(* IEC 61131-3 sources: Mizera_Tube/Plc (part 5) *)

(* ---- usrCh8.plc ---- *)
*******************************************************************************
*******************************************************************************
*   @@@ CH8: Unload machine management
*******************************************************************************
*******************************************************************************
#funcdec "assi.plc"
#funcdec "cnc.plc"

#include "usrMem.inc"

VAR_IN_OUT
#include "mem.inc"
END_VAR

VAR
#include "cnc.inc"

GESTCH8:            GESTCH;
CH8END:             GESTCHEND;
GESTAX70:           GESTAX;
GESTAX71:           GESTAX;                         * Saw Following Support
GESTAX72:           GESTAX;
GESTAX73:           GESTAX;
GESTAX74:           GESTAX;
GESTAX75:           GESTAX;
AXLSREF71:          AX_LS_REF;
AXLSREF72:          AX_LS_REF;
AXLSREF73:          AX_LS_REF;
AXLSREF74:          AX_LS_REF;
AXLSREF75:          AX_LS_REF;

RTRIG_AX_SEL71:     R_TRIG;
RTRIG_AX_SEL72:     R_TRIG;
RTRIG_AX_SEL73:     R_TRIG;
RTRIG_AX_SEL74:     R_TRIG;
RTRIG_AX_SEL75:     R_TRIG;

UnSupp_71_GoUp:    BOOL;
UnSupp_72_GoUp:    BOOL;
UnSupp_73_GoUp:    BOOL;
UnSupp_74_GoUp:    BOOL;
UnSupp_75_GoUp:    BOOL;

END_VAR

#include "iol.inc"

VAR_IN_OUT
#include "usrIol.inc"
ActualQtaAbsRef     AT %pa18;                       * Absolute homing quota
QtaRefAbsSet        AT %LsPlc50;                    * Absolute homing quota setting
END_VAR

FUNCTION CH8

PATH %cn8

LD   ALWAYS_ONE                                     ** PLCFLAGS.1  Flag sempre stato on
ST   GESTCH8.xCmdFromInput

LD   ALWAYS_ONE                                     ** PLCFLAGS.1  Flag sempre stato on
ST   GESTCH8.xEscOpCmd

LD   %PLCFLAGS.0
ST   GESTCH8.xSelFromInput                          * Disabilita selezioni standard macchina

LD   Ch0_Ref_Gen
ST   GESTCH8.xSelREF

LD   Ch0_Ref_Sin
ST   GESTCH8.xSingleRef

LD   Ch0_Jog
ST   GESTCH8.xSelJOG

LD   Ch0_Inc
ST   GESTCH8.xSelINC

LD   Ch0_Auto
ST   GESTCH8.xSelAUT

LD   ProgRunCh0
ANDN %cn0.rc8.1
ANDN PlcEmerGen                                     ** M0.10 Emergenza generale
OR (
LD   Start_Ch0
AND  ch8_in_ref
)
OR(
LD   Start_Ch0
AND  BCI_MDI                                        ** rc0.11  Selettore modi operativi su MDI (semiautom)
AND (
 LD  UP_SELCHAN                                     ** ui17 Canale selezionato da monitor canale
 EQ  8
)
)
ST   GESTCH8.xStart                                 * comando START al canale (esterno)

LD   ResetChannels
ST   GESTCH8.xReset                                 * comando RESET al canale (esterno)

LD   %cn0.rc8.1                                    ** Condizioni richiesta hold canale 0
OR(
LD   Pul_Stop_Req
AND  BCI_MDI                                        ** rc0.11  Selettore modi operativi su MDI (semiautom)
)
ST   GESTCH8.xHold                                  * comando Hold al canale (esterno)

LD   Ch0Alarm
ST   GESTCH8.xEmer                                  * comando Emergenza al canale (esterno)

LD   8888
ST   GESTCH8.xPPNumber                              * numero part program da eseguire

LD   %PLCFLAGS.0
ST   GESTCH8.xBlkSearch
ST   GESTCH8.xIntBlkSrc                             * Forzam. esec. ricerca blocco interna
ST   GESTCH8.xOverstore                             * Ab. overstore dopo ricerca blocco (provv.)

LD   MainChFeedrate                                 ** feedrate for channel
ST   GESTCH8.xOverride

CAL  GESTCH8

LD   GESTCH8.yProgramRun                            * Programma in corso
ST   PRGRUN_CN8

LD   BCO_STB_GET                                    ** rc8.17 Strobe per GET resources
AND  AxStopSincGRPMacc                              ** (gPlc13.11)Assi Fermi per sincronismo GRP[ax]
ST   BCI_ACK_GET                                    ** rc0.29  ACK per GET resource

********************************************************************************
* Unload axes
********************************************************************************
* Virtual Axis(70)

LD  %cc1.0                                          * Maschera assi associata al canale 8
JMPCN noAx70

PATH %ax70

LD   ALWAYS_ZERO
ST   GESTAX70.xJogPlus

LD   ALWAYS_ZERO
ST   GESTAX70.xJogMinus

LD   ALWAYS_ONE
ST   GESTAX70.xZeroForced                           * Forzamento asse tarato

LD   ALWAYS_ZERO
ST   GESTAX70.xHoldMoving                           * Richiesta blocco avanzamento

LD   Res_Axes                                       ** (gPlc25.1) reset axes disable electric shaft
ST   GESTAX70.xUnlock

LDN  ch8_in_ref                                     ** channel 3 in ref
ST   GESTAX70.xEnFIR                                * Abilita filtri FIR
ST   GESTAX70.xEnFrComp                             ** Abilita friction compensation

LD   ALWAYS_ZERO                                    ** PLCFLAGS.0  Flag sempre stato off
ST   GESTAX70.xDisLimiter

LD   GESTAX50_xCloseLoop
ST   GESTAX70.xCloseLoop

LD   %cn0.rc8.3                                     * ch0 in alarm
OR   %cn3.rc8.3                                     * ch3 in alarm
**OR   EmerINC
ST   GESTAX70.xSetAlarm                             ** Forzamento allarme asse

CAL  GESTAX70

noAx70:

********************************************************************************
* Unload Support for Saw Cutting (71)
********************************************************************************
PATH %ax71
PATH %ax_lsref71

***************************************
*   POWER ON (PON)
***************************************
LD   %pa3.31                                        * Simulato
ORN  %cc1.1                                         * Maschera assi associata al canale
OR(
LD   %nvel11                                        ** 3,4=CANopen, Ecat
EQ   3
)
OR(
LD   %nvel11                                        ** 3,4=CANopen, Ecat
EQ   4
)
ST   Pon_UnSupp_71                                  ** PON unload support axis
***************************************

LDN  %ra3.2                                         * ra3.2  Direzione moto asse avanti
OR   %ra0.9                                         * ra0.9 Comando indietro
AND  %ra3.13                                        * ra3.13  Ordine di moto
ST   UnSupp_71_GoUp

LD  %cc1.1                                          * Maschera assi associata al canale 8
JMPCN NOAX71

***
*   LIMIT SWITCH & REFERENCE SWITCH

LD   %lsrefmode
ST   AXLSREF71.x_REF_mode                           * 0=use ref switch...

LD   %lsreflevel
ST   AXLSREF71.x_TYPE_LS                            * (1=NC, 0=NO)

LD   I_I_FC_L1_NEG
ST   AXLSREF71.x_MIN_LS                             * Min Limit switch

LD   I_I_FC_L1_POS                * C saw minimumm limit switchV
ST   AXLSREF71.x_MAX_LS                             * Max Limit switch

LD   ALWAYS_ZERO
ST   AXLSREF71.x_REF_S                              * Reference switch

CAL  AXLSREF71

LD   AXLSREF71.y_MIN_LS                             * Min Limit switch
ST   GESTAX71.xMinusLS                              * Negative limit switch

LD   AXLSREF71.y_MAX_LS                             * Max Limit switch
ST   GESTAX71.xPlusLS                               * Positive limit switch

LD   AXLSREF71.y_REF_S                              * Reference switch
ST   GESTAX71.xRefLS                                * Reference
***

LD   MainAxesPowerAllowed
AND  MainAxesPower                                  * PON
ST   GESTAX71.xCloseLoop

LD   GstMaccSelYCh8
ST   GESTAX71.xSelected

***************************************
* Change REF quota for ABS reference
***************************************
CAL  RTRIG_AX_SEL71(CLK:=GESTAX71.xSelected)

LD   RTRIG_AX_SEL71.Q
JMPCN NoSel71
LD   ActualQtaAbsRef                                ** Absolute homing quota
ST   QtaRefAbsSet                                   ** Absolute homing quota setting
NoSel71:

LD   GESTAX71.xSelected
AND  %nvel14.0                                      * Se Vale 1 ?gestito "Encoder Assoluto" (Da Configura Asse)
AND (
LD   ActualQtaAbsRef                                ** Absolute homing quota
NE   QtaRefAbsSet                                   ** Absolute homing quota setting
)
JMPCN NoEq71

LD   QtaRefAbsSet                                   ** Absolute homing quota setting
ST   ActualQtaAbsRef                                ** Absolute homing quota
NoEq71:
***************************************

LD   Pul_Jogp                                       ** (gPlc0.4)jog+ pushbutton
AND  GESTAX71.xSelected
ANDN PlcEmerGen                                     ** M0.10 Emergenza generale
AND  GESTAX71.xCloseLoop
ST   GESTAX71.xJogPlus

LD   Pul_Jogm                                       ** (gPlc0.5)jog- pushbutton
AND  GESTAX71.xSelected
ANDN PlcEmerGen                                     ** M0.10 Emergenza generale
AND  GESTAX71.xCloseLoop
ANDN CMD_HOLDMOVING_CH8.1
ST   GESTAX71.xJogMinus

LD   %nvel14.0                                      * Se Vale 1 ?gestito "Encoder Assoluto" (Da Configura Asse)
ST   GESTAX71.xZeroForced                           * Forzamento asse tarato

LD   GESTAX2_xHoldMoving                            * Richiesta blocco avanzamento
OR   CMD_HOLDMOVING_CH8.1                           ** M203 Hold moving command axis CH5 (bit0=X, bit1=Y...)
ST   GESTAX71.xHoldMoving                           * Richiesta blocco avanzamento

LD   Res_Axes                                       ** (gPlc25.1) reset axes disable electric shaft
ST   GESTAX71.xUnlock

LDN  ch8_in_ref                                     ** channel 3 in ref
ST   GESTAX71.xEnFIR                                * Abilita filtri FIR
ST   GESTAX71.xEnFrComp                             ** Abilita friction compensation

LD   ALWAYS_ZERO                                    ** PLCFLAGS.0  Flag sempre stato off
ST   GESTAX71.xDisLimiter

LD   %cn0.rc8.3                                     * ch0 in alarm
OR   %cn3.rc8.3                                     * ch3 in alarm
**OR   EmerINC
ST   GESTAX71.xSetAlarm                             ** Forzamento allarme asse

LD   usrReqGrantSup1
ST   GESTAX71.xFromPlc

CAL  GESTAX71

LD   GESTAX71.yDriveNotEn
S    %PLCerr3.0                                     * Axis 71, drive not enable

LD   BSG_INC                                        ** rg1.2 Selezione modo INC (inc.fissi)
JMPCN SVIX71

LD   %pa59                                          * Velocit?di Repos
MUL  1000
DIV  60
MUL  MainChFeedrate                                 ** (gPlc16) feed degli assi (%)
DIV  100
ST   %ra50                                          * Limitazione velocita' massima interpolazione

SVIX71:
NOAX71:

********************************************************************************
* Unload Support 1 (ax72)
********************************************************************************
PATH %ax72
PATH %ax_lsref72

***************************************
*   POWER ON (PON)
***************************************
LD   %pa3.31            * Simulato
ORN  %cc1.2             * Maschera assi associata al canale
OR(
LD   %nvel11            ** 3,4=CANopen, Ecat
EQ   3
)
OR(
LD   %nvel11            ** 3,4=CANopen, Ecat
EQ   4
)
ST   Pon_UnSupp_72      ** PON unload support axis
***************************************

LDN  %ra3.2                                         * ra3.2  Direzione moto asse avanti
OR   %ra0.9                                         * ra0.9 Comando indietro
AND  %ra3.13                                        * ra3.13  Ordine di moto
ST   UnSupp_72_GoUp

LD  %cc1.2           * Maschera assi associata al canale 8
JMPCN NOAX72

***
*   LIMIT SWITCH & REFERENCE SWITCH

LD   %lsrefmode
ST   AXLSREF72.x_REF_mode        * 0=use ref switch...

LD   %lsreflevel
ST   AXLSREF72.x_TYPE_LS         * (1=NC, 0=NO)

LD   I_I_FC_L2_NEG
ST   AXLSREF72.x_MIN_LS          * Min Limit switch

LD   I_I_FC_L2_POS               * C saw maximun limit switch
ST   AXLSREF72.x_MAX_LS          * Max Limit switch

LD   ALWAYS_ZERO
ST   AXLSREF72.x_REF_S           * Reference switch

CAL  AXLSREF72

LD   AXLSREF72.y_MIN_LS          * Min Limit switch
ST   GESTAX72.xMinusLS           * Negative limit switch

LD   AXLSREF72.y_MAX_LS          * Max Limit switch
ST   GESTAX72.xPlusLS            * Positive limit switch

LD   AXLSREF72.y_REF_S           * Reference switch
ST   GESTAX72.xRefLS             * Reference
***

LD   MainAxesPowerAllowed
AND  MainAxesPower               * PON
ST   GESTAX72.xCloseLoop

LD   GstMaccSelZCh8
ST   GESTAX72.xSelected

***************************************
* Change REF quota for ABS reference
***************************************
CAL  RTRIG_AX_SEL72(CLK:=GESTAX72.xSelected)

LD   RTRIG_AX_SEL72.Q
JMPCN NoSel72
LD   ActualQtaAbsRef               ** Absolute homing quota
ST   QtaRefAbsSet                  ** Absolute homing quota setting
NoSel72:

LD   GESTAX72.xSelected
AND  %nvel14.0                     * Se Vale 1 � gestito "Encoder Assoluto" (Da Configura Asse)
AND (
LD   ActualQtaAbsRef               ** Absolute homing quota
NE   QtaRefAbsSet                  ** Absolute homing quota setting
)
JMPCN NoEq72

LD   QtaRefAbsSet                  ** Absolute homing quota setting
ST   ActualQtaAbsRef               ** Absolute homing quota
NoEq72:
***************************************

LD   Pul_Jogp                      ** (gPlc0.4)jog+ pushbutton
AND  GESTAX72.xSelected
ANDN PlcEmerGen                      ** M0.10 Emergenza generale
AND  GESTAX72.xCloseLoop
ST   GESTAX72.xJogPlus

LD   Pul_Jogm                      ** (gPlc0.5)jog- pushbutton
AND  GESTAX72.xSelected
ANDN PlcEmerGen                      ** M0.10 Emergenza generale
AND  GESTAX72.xCloseLoop
ANDN CMD_HOLDMOVING_CH8.2
ST   GESTAX72.xJogMinus

LD   %nvel14.0                     * Se Vale 1 � gestito "Encoder Assoluto" (Da Configura Asse)
ST   GESTAX72.xZeroForced          * Forzamento asse tarato

LD   GESTAX2_xHoldMoving           * Richiesta blocco avanzamento
OR   CMD_HOLDMOVING_CH8.2          ** M203 Hold moving command axis CH5 (bit0=X, bit1=Y...)
ST   GESTAX72.xHoldMoving          * Richiesta blocco avanzamento

LD   Res_Axes                      ** (gPlc25.1) reset axes disable electric shaft
ST   GESTAX72.xUnlock

LDN  ch8_in_ref                    ** channel 3 in ref
ST   GESTAX72.xEnFIR               * Abilita filtri FIR
ST   GESTAX72.xEnFrComp            ** Abilita friction compensation

LD   ALWAYS_ZERO                   ** PLCFLAGS.0  Flag sempre stato off
ST   GESTAX72.xDisLimiter

LD   %cn0.rc8.3                    * ch0 in alarm
OR   %cn3.rc8.3                    * ch3 in alarm
ST   GESTAX72.xSetAlarm            ** Forzamento allarme asse

LD   usrReqGrantSup2
ST   GESTAX72.xFromPlc

CAL  GESTAX72

LD   GESTAX72.yDriveNotEn
S    %PLCerr3.1                    * Axis 72, drive not enable

LD   BSG_INC                       ** rg1.2 Selezione modo INC (inc.fissi)
JMPCN SVIX72

LD   %pa59                         * Velocit� di Repos
MUL  1000
DIV  60
MUL  MainChFeedrate                ** (gPlc16) feed degli assi (%)
DIV  100
ST   %ra50                         * Limitazione velocita' massima interpolazione

SVIX72:
NOAX72:

********************************************************************************
* Unload Support 2 (ax73)
********************************************************************************
PATH %ax73
PATH %ax_lsref73

***************************************
*   POWER ON (PON)
***************************************
LD   %pa3.31                                        * Simulato
ORN  %cc1.3                                         * Maschera assi associata al canale
OR(
LD   %nvel11                                        ** 3,4=CANopen, Ecat
EQ   3
)
OR(
LD   %nvel11                                        ** 3,4=CANopen, Ecat
EQ   4
)
ST   Pon_UnSupp_73                                  ** PON unload support axis
***************************************

LDN  %ra3.2                                         * ra3.2  Direzione moto asse avanti
OR   %ra0.9                                         * ra0.9 Comando indietro
AND  %ra3.13                                        * ra3.13  Ordine di moto
ST   UnSupp_73_GoUp

LD  %cc1.3                                          * Maschera assi associata al canale 8
JMPCN NOAX73

***
*   LIMIT SWITCH & REFERENCE SWITCH

LD   %lsrefmode
ST   AXLSREF73.x_REF_mode                           * 0=use ref switch...

LD   %lsreflevel
ST   AXLSREF73.x_TYPE_LS                            * (1=NC, 0=NO)

LD   I_I_FC_L3_NEG
ST   AXLSREF73.x_MIN_LS                             * Min Limit switch

LD   I_I_FC_L3_POS                                  * W maximun limit switch
ST   AXLSREF73.x_MAX_LS                             * Max Limit switch

LD   ALWAYS_ZERO
ST   AXLSREF73.x_REF_S                              * Reference switch

CAL  AXLSREF73

LD   AXLSREF73.y_MIN_LS                             * Min Limit switch
ST   GESTAX73.xMinusLS                              * Negative limit switch

LD   AXLSREF73.y_MAX_LS                             * Max Limit switch
ST   GESTAX73.xPlusLS                               * Positive limit switch

LD   AXLSREF73.y_REF_S                              * Reference switch
ST   GESTAX73.xRefLS                                * Reference
***

LD   MainAxesPowerAllowed
AND  MainAxesPower                                  * PON
ST   GESTAX73.xCloseLoop

LD   GstMaccSelUCh8
ST   GESTAX73.xSelected

***************************************
* Change REF quota for ABS reference
***************************************
CAL  RTRIG_AX_SEL73(CLK:=GESTAX73.xSelected)

LD   RTRIG_AX_SEL73.Q
JMPCN NoSel73
LD   ActualQtaAbsRef                                ** Absolute homing quota
ST   QtaRefAbsSet                                   ** Absolute homing quota setting
NoSel73:

LD   GESTAX73.xSelected
AND  %nvel14.0                                      * Se Vale 1 ?gestito "Encoder Assoluto" (Da Configura Asse)
AND (
LD   ActualQtaAbsRef                                ** Absolute homing quota
NE   QtaRefAbsSet                                   ** Absolute homing quota setting
)
JMPCN NoEq73

LD   QtaRefAbsSet                                   ** Absolute homing quota setting
ST   ActualQtaAbsRef                                ** Absolute homing quota
NoEq73:
***************************************

LD   Pul_Jogp                                       ** (gPlc0.4)jog+ pushbutton
AND  GESTAX73.xSelected
ANDN PlcEmerGen                                     ** M0.10 Emergenza generale
AND  GESTAX73.xCloseLoop
ST   GESTAX73.xJogPlus

LD   Pul_Jogm                                       ** (gPlc0.5)jog- pushbutton
AND  GESTAX73.xSelected
ANDN PlcEmerGen                                     ** M0.10 Emergenza generale
AND  GESTAX73.xCloseLoop
ANDN CMD_HOLDMOVING_CH8.3
ST   GESTAX73.xJogMinus

LD   %nvel14.0                                      * Se Vale 1 ?gestito "Encoder Assoluto" (Da Configura Asse)
ST   GESTAX73.xZeroForced                           * Forzamento asse tarato

LD   GESTAX2_xHoldMoving                            * Richiesta blocco avanzamento
OR  CMD_HOLDMOVING_CH8.3                           ** M203 Hold moving command axis CH5 (bit0=X, bit1=Y...)
ST   GESTAX73.xHoldMoving                           * Richiesta blocco avanzamento

LD   Res_Axes                                       ** (gPlc25.1) reset axes disable electric shaft
ST   GESTAX73.xUnlock

LDN  ch8_in_ref                                     ** channel 3 in ref
ST   GESTAX73.xEnFIR                                * Abilita filtri FIR
ST   GESTAX73.xEnFrComp                             ** Abilita friction compensation

LD   ALWAYS_ZERO                                    ** PLCFLAGS.0  Flag sempre stato off
ST   GESTAX73.xDisLimiter

LD   %cn0.rc8.3                                     * ch0 in alarm
OR   %cn3.rc8.3                                     * ch3 in alarm
**OR   EmerINC
ST   GESTAX73.xSetAlarm                             ** Forzamento allarme asse

LD   usrReqGrantSup3
ST   GESTAX73.xFromPlc

CAL  GESTAX73

LD   GESTAX73.yDriveNotEn
S    %PLCerr3.2                                     * Axis 73, drive not enable

LD   BSG_INC                                        ** rg1.2 Selezione modo INC (inc.fissi)
JMPCN SVIX73

LD   %pa59                                          * Velocit?di Repos
MUL  1000
DIV  60
MUL  MainChFeedrate                                 ** (gPlc16) feed degli assi (%)
DIV  100
ST   %ra50                                          * Limitazione velocita' massima interpolazione

SVIX73:
NOAX73:

********************************************************************************
* Unload Support 3 (ax74)
********************************************************************************
PATH %ax74
PATH %ax_lsref74

***************************************
*   POWER ON (PON)
***************************************
LD   %pa3.31                                        * Simulato
ORN  %cc1.4                                         * Maschera assi associata al canale
OR(
LD   %nvel11                                        ** 3,4=CANopen, Ecat
EQ   3
)
OR(
LD   %nvel11                                        ** 3,4=CANopen, Ecat
EQ   4
)
ST   Pon_UnSupp_74                                  ** PON unload support axis
***************************************

LDN  %ra3.2                                         * ra3.2  Direzione moto asse avanti
OR   %ra0.9                                         * ra0.9 Comando indietro
AND  %ra3.13                                        * ra3.13  Ordine di moto
ST   UnSupp_74_GoUp

LD  %cc1.4                                          * Maschera assi associata al canale 8
JMPCN NOAX74

***
*   LIMIT SWITCH & REFERENCE SWITCH

LD   %lsrefmode
ST   AXLSREF74.x_REF_mode                           * 0=use ref switch...

LD   %lsreflevel
ST   AXLSREF74.x_TYPE_LS                            * (1=NC, 0=NO)

LD   I_I_FC_L4_NEG
ST   AXLSREF74.x_MIN_LS                             * Min Limit switch

LD   I_I_FC_L4_POS                                  * W minimumm limit switch
ST   AXLSREF74.x_MAX_LS                             * Max Limit switch

LD   ALWAYS_ZERO
ST   AXLSREF74.x_REF_S                              * Reference switch

CAL  AXLSREF74

LD   AXLSREF74.y_MIN_LS                             * Min Limit switch
ST   GESTAX74.xMinusLS                              * Negative limit switch

LD   AXLSREF74.y_MAX_LS                             * Max Limit switch
ST   GESTAX74.xPlusLS                               * Positive limit switch

LD   AXLSREF74.y_REF_S                              * Reference switch
ST   GESTAX74.xRefLS                                * Reference
***

LD   MainAxesPowerAllowed
AND  MainAxesPower                                  * PON
ST   GESTAX74.xCloseLoop

LD   GstMaccSelVCh8
ST   GESTAX74.xSelected

***************************************
* Change REF quota for ABS reference
***************************************
CAL  RTRIG_AX_SEL74(CLK:=GESTAX74.xSelected)

LD   RTRIG_AX_SEL74.Q
JMPCN NoSel74
LD   ActualQtaAbsRef                                ** Absolute homing quota
ST   QtaRefAbsSet                                   ** Absolute homing quota setting
NoSel74:

LD   GESTAX74.xSelected
AND  %nvel14.0                                      * Se Vale 1 ?gestito "Encoder Assoluto" (Da Configura Asse)
AND (
LD   ActualQtaAbsRef                                ** Absolute homing quota
NE   QtaRefAbsSet                                   ** Absolute homing quota setting
)
JMPCN NoEq74

LD   QtaRefAbsSet                                   ** Absolute homing quota setting
ST   ActualQtaAbsRef                                ** Absolute homing quota
NoEq74:
***************************************

LD   Pul_Jogp                                       ** (gPlc0.4)jog+ pushbutton
AND  GESTAX74.xSelected
ANDN PlcEmerGen                                     ** M0.10 Emergenza generale
AND  GESTAX74.xCloseLoop
ST   GESTAX74.xJogPlus

LD   Pul_Jogm                                       ** (gPlc0.5)jog- pushbutton
AND  GESTAX74.xSelected
ANDN PlcEmerGen                                     ** M0.10 Emergenza generale
AND  GESTAX74.xCloseLoop
ANDN CMD_HOLDMOVING_CH8.4
ST   GESTAX74.xJogMinus

LD   %nvel14.0                                      * Se Vale 1 ?gestito "Encoder Assoluto" (Da Configura Asse)
ST   GESTAX74.xZeroForced                           * Forzamento asse tarato

LD   GESTAX2_xHoldMoving                            * Richiesta blocco avanzamento
OR   CMD_HOLDMOVING_CH8.4                           ** M203 Hold moving command axis CH5 (bit0=X, bit1=Y...)
ST   GESTAX74.xHoldMoving                           * Richiesta blocco avanzamento

LD   Res_Axes                                       ** (gPlc25.1) reset axes disable electric shaft
ST   GESTAX74.xUnlock

LDN  ch8_in_ref                                     ** channel 3 in ref
ST   GESTAX74.xEnFIR                                * Abilita filtri FIR
ST   GESTAX74.xEnFrComp                             ** Abilita friction compensation

LD   ALWAYS_ZERO                                    ** PLCFLAGS.0  Flag sempre stato off
ST   GESTAX74.xDisLimiter

LD   %cn0.rc8.3                                     * ch0 in alarm
OR   %cn3.rc8.3                                     * ch3 in alarm
ST   GESTAX74.xSetAlarm                             ** Forzamento allarme asse

LD   usrReqGrantSup4
ST   GESTAX74.xFromPlc

CAL  GESTAX74

LD   GESTAX74.yDriveNotEn
S    %PLCerr3.3                                     * Axis 74, drive not enable

LD   BSG_INC                                        ** rg1.2 Selezione modo INC (inc.fissi)
JMPCN SVIX74

LD   %pa59                                          * Velocit?di Repos
MUL  1000
DIV  60
MUL  MainChFeedrate                                 ** (gPlc16) feed degli assi (%)
DIV  100
ST   %ra50                                          * Limitazione velocita' massima interpolazione

SVIX74:
NOAX74:

********************************************************************************
* Unload Support 4 (ax75)
********************************************************************************
PATH %ax75
PATH %ax_lsref75

***************************************
*   POWER ON (PON)
***************************************
LD   %pa3.31                                        * Simulato
ORN  %cc1.5                                         * Maschera assi associata al canale
OR(
LD   %nvel11                                        ** 3,4=CANopen, Ecat
EQ   3
)
OR(
LD   %nvel11                                        ** 3,4=CANopen, Ecat
EQ   4
)
ST   Pon_UnSupp_75                                  ** PON unload support axis
***************************************

LDN  %ra3.2                                         * ra3.2  Direzione moto asse avanti
OR   %ra0.9                                         * ra0.9 Comando indietro
AND  %ra3.13                                        * ra3.13  Ordine di moto
ST   UnSupp_75_GoUp

LD  %cc1.5                                          * Maschera assi associata al canale 8
JMPCN NOAX75

***
*   LIMIT SWITCH & REFERENCE SWITCH

LD   %lsrefmode
ST   AXLSREF75.x_REF_mode                           * 0=use ref switch...

LD   %lsreflevel
ST   AXLSREF75.x_TYPE_LS                            * (1=NC, 0=NO)

LD   I_I_FC_L5_NEG
ST   AXLSREF75.x_MIN_LS                             * Min Limit switch

LD   I_I_FC_L5_POS
ST   AXLSREF75.x_MAX_LS                             * Max Limit switch

LD   ALWAYS_ZERO
ST   AXLSREF75.x_REF_S                              * Reference switch

CAL  AXLSREF75

LD   AXLSREF75.y_MIN_LS                             * Min Limit switch
ST   GESTAX75.xMinusLS                              * Negative limit switch

LD   AXLSREF75.y_MAX_LS                             * Max Limit switch
ST   GESTAX75.xPlusLS                               * Positive limit switch

LD   AXLSREF75.y_REF_S                              * Reference switch
ST   GESTAX75.xRefLS                                * Reference
***

LD   MainAxesPowerAllowed
AND  MainAxesPower                                  * PON
ST   GESTAX75.xCloseLoop

LD   GstMaccSelWCh8
ST   GESTAX75.xSelected

***************************************
* Change REF quota for ABS reference
***************************************
CAL  RTRIG_AX_SEL75(CLK:=GESTAX75.xSelected)

LD   RTRIG_AX_SEL75.Q
JMPCN NoSel75
LD   ActualQtaAbsRef                                ** Absolute homing quota
ST   QtaRefAbsSet                                   ** Absolute homing quota setting
NoSel75:

LD   GESTAX75.xSelected
AND  %nvel14.0                                      * Se Vale 1 ?gestito "Encoder Assoluto" (Da Configura Asse)
AND (
LD   ActualQtaAbsRef                                ** Absolute homing quota
NE   QtaRefAbsSet                                   ** Absolute homing quota setting
)
JMPCN NoEq75

LD   QtaRefAbsSet                                   ** Absolute homing quota setting
ST   ActualQtaAbsRef                                ** Absolute homing quota
NoEq75:
***************************************

LD   Pul_Jogp                                       ** (gPlc0.4)jog+ pushbutton
AND  GESTAX75.xSelected
ANDN PlcEmerGen                                     ** M0.10 Emergenza generale
AND  GESTAX75.xCloseLoop
ST   GESTAX75.xJogPlus

LD   Pul_Jogm                                       ** (gPlc0.5)jog- pushbutton
AND  GESTAX75.xSelected
ANDN PlcEmerGen                                     ** M0.10 Emergenza generale
AND  GESTAX75.xCloseLoop
ANDN CMD_HOLDMOVING_CH8.5
ST   GESTAX75.xJogMinus

LD   %nvel14.0                                      * Se Vale 1 ?gestito "Encoder Assoluto" (Da Configura Asse)
ST   GESTAX75.xZeroForced                           * Forzamento asse tarato

LD   GESTAX2_xHoldMoving                           * Richiesta blocco avanzamento
OR   CMD_HOLDMOVING_CH8.5                           ** M203 Hold moving command axis CH5 (bit0=X, bit1=Y...)
ST   GESTAX75.xHoldMoving                           * Richiesta blocco avanzamento

LD   Res_Axes                                       ** (gPlc25.1) reset axes disable electric shaft
ST   GESTAX75.xUnlock

LDN  ch8_in_ref                                     ** channel 3 in ref
ST   GESTAX75.xEnFIR                                * Abilita filtri FIR
ST   GESTAX75.xEnFrComp                             ** Abilita friction compensation

LD   ALWAYS_ZERO                                    ** PLCFLAGS.0  Flag sempre stato off
ST   GESTAX75.xDisLimiter

LD   %cn0.rc8.3                                     * ch0 in alarm
OR   %cn3.rc8.3                                     * ch3 in alarm
**OR   EmerINC
ST   GESTAX75.xSetAlarm                             ** Forzamento allarme asse

LD   usrReqGrantSup5
ST   GESTAX75.xFromPlc

CAL  GESTAX75

LD   GESTAX75.yDriveNotEn
S    %PLCerr3.3                                     * Axis 75, drive not enable

LD   BSG_INC                                        ** rg1.2 Selezione modo INC (inc.fissi)
JMPCN SVIX75

LD   %pa59                                          * Velocit?di Repos
MUL  1000
DIV  60
MUL  MainChFeedrate                                 ** (gPlc16) feed degli assi (%)
DIV  100
ST   %ra50                                          * Limitazione velocita' massima interpolazione

SVIX75:
NOAX75:

**************************
* Acknowledg funzioni "M"
**************************
*
LD   %PLCFLAGS.0
ST   CH8END.xWaitMFun

CAL  CH8END

END_FUNCTION

(* ---- usrCh9.plc ---- *)
*******************************************************************************
*******************************************************************************
*   @@@ CH9: Lateral /Loader horizontal axes support
*******************************************************************************
*******************************************************************************
#funcdec "assi.plc"
#funcdec "cnc.plc"

#include "usrMem.inc"

VAR_IN_OUT
#include "mem.inc"
END_VAR

VAR
#include "cnc.inc"

GESTCH9:            GESTCH;
CH9END:             GESTCHEND;
GESTAX80:           GESTAX;    * virtual axes for following
GESTAX81:           GESTAX;
GESTAX82:           GESTAX;
GESTAX83:           GESTAX;
GESTAX84:           GESTAX;

AXLSREF81:          AX_LS_REF;
AXLSREF82:          AX_LS_REF;
AXLSREF83:          AX_LS_REF;
AXLSREF84:          AX_LS_REF;
AXLSREF85:          AX_LS_REF;

RTRIG_AX_SEL81:     R_TRIG;
RTRIG_AX_SEL82:     R_TRIG;
RTRIG_AX_SEL83:     R_TRIG;
RTRIG_AX_SEL84:     R_TRIG;
RTRIG_AX_SEL85:     R_TRIG;

UnSupp_81_GoUp:    BOOL;
UnSupp_82_GoUp:    BOOL;
UnSupp_83_GoUp:    BOOL;
UnSupp_84_GoUp:    BOOL;
UnSupp_85_GoUp:    BOOL;

END_VAR

#include "iol.inc"

VAR_IN_OUT
#include "usrIol.inc"
ActualQtaAbsRef     AT %pa18;                       * Absolute homing quota
QtaRefAbsSet        AT %LsPlc50;                    * Absolute homing quota setting

END_VAR

FUNCTION CH9

PATH %cn9

LD   ALWAYS_ONE                                     ** PLCFLAGS.1  Flag sempre stato on
ST   GESTCH9.xCmdFromInput

LD   ALWAYS_ONE                                     ** PLCFLAGS.1  Flag sempre stato on
ST   GESTCH9.xEscOpCmd

LD   %PLCFLAGS.0
ST   GESTCH9.xSelFromInput                          * Disabilita selezioni standard macchina

LD   Ch0_Ref_Gen
ST   GESTCH9.xSelREF

LD   Ch0_Ref_Sin
ST   GESTCH9.xSingleRef

LD   Ch0_Jog
ST   GESTCH9.xSelJOG

LD   Ch0_Inc
ST   GESTCH9.xSelINC

LD   Ch0_Auto
ST   GESTCH9.xSelAUT

LD   %PLCFLAGS.0                                    ** Condizioni richiesta hold canale 0
ST   GESTCH9.xStart                                 * comando START al canale (esterno)

LD   ResetChannels
ST   GESTCH9.xReset                                 * comando RESET al canale (esterno)

LD   %PLCFLAGS.0                                    ** Condizioni richiesta hold canale 0
OR(
LD   Pul_Stop_Req
AND  BCI_MDI                                        ** rc0.11  Selettore modi operativi su MDI (semiautom)
)
ST   GESTCH9.xHold                                  * comando Hold al canale (esterno)

LD   Ch0Alarm
ST   GESTCH9.xEmer                                  * comando Emergenza al canale (esterno)

LD   99999
ST   GESTCH9.xPPNumber                              * numero part program da eseguire

LD   %PLCFLAGS.0
ST   GESTCH9.xBlkSearch
ST   GESTCH9.xIntBlkSrc                             * Forzam. esec. ricerca blocco interna
ST   GESTCH9.xOverstore                             * Ab. overstore dopo ricerca blocco (provv.)

LD   MainChFeedrate                                 ** feedrate for channel
ST   GESTCH9.xOverride

CAL  GESTCH9

LD   GESTCH9.yProgramRun                            * Programma in corso
ST   PRGRUN_CN9

LD   BCO_STB_GET                                    ** rc8.17 Strobe per GET resources
AND  AxStopSincGRPMacc                              ** (gPlc13.11)Assi Fermi per sincronismo GRP[ax]
ST   BCI_ACK_GET                                    ** rc0.29  ACK per GET resource

********************************************************************************
* Unload axes
********************************************************************************
* Virtual Axis(70)

LD  %cc1.0                                          * Maschera assi associata al canale 8
JMPCN noAx80

PATH %ax80

LD   ALWAYS_ZERO
ST   GESTAX80.xJogPlus

LD   ALWAYS_ZERO
ST   GESTAX80.xJogMinus

LD   ALWAYS_ONE
ST   GESTAX80.xZeroForced                           * Forzamento asse tarato

LD   ALWAYS_ZERO
ST   GESTAX80.xHoldMoving                           * Richiesta blocco avanzamento

LD   Res_Axes                                       ** (gPlc25.1) reset axes disable electric shaft
ST   GESTAX80.xUnlock

LDN  ch9_in_ref                                     ** channel 3 in ref
ST   GESTAX80.xEnFIR                                * Abilita filtri FIR
ST   GESTAX80.xEnFrComp                             ** Abilita friction compensation

LD   ALWAYS_ZERO                                    ** PLCFLAGS.0  Flag sempre stato off
ST   GESTAX80.xDisLimiter

LD   GESTAX50_xCloseLoop
ST   GESTAX80.xCloseLoop

LD   %cn0.rc8.3                                     * ch0 in alarm
OR   %cn3.rc8.3                                     * ch3 in alarm
**OR   EmerINC
ST   GESTAX80.xSetAlarm                             ** Forzamento allarme asse

CAL  GESTAX80

noAx80:

********************************************************************************
* Unload Support for Saw Cutting (81) 2
********************************************************************************
PATH %ax81
PATH %ax_lsref81

***************************************
*   POWER ON (PON)
***************************************
LD   %pa3.31                                        * Simulato
ORN  %cc1.1                                         * Maschera assi associata al canale
OR(
LD   %nvel11                                        ** 3,4=CANopen, Ecat
EQ   3
)
OR(
LD   %nvel11                                        ** 3,4=CANopen, Ecat
EQ   4
)
ST   Pon_UnSupp_81                                  ** PON unload support axis
***************************************

LDN  %ra3.2                                         * ra3.2  Direzione moto asse avanti
OR   %ra0.9                                         * ra0.9 Comando indietro
AND  %ra3.13                                        * ra3.13  Ordine di moto
ST   UnSupp_81_GoUp

LD  %cc1.1                                          * Maschera assi associata al canale 8
JMPCN NOAX81

***
*   LIMIT SWITCH & REFERENCE SWITCH

LD   %lsrefmode
ST   AXLSREF81.x_REF_mode                           * 0=use ref switch...

LD   %lsreflevel
ST   AXLSREF81.x_TYPE_LS                            * (1=NC, 0=NO)

LD   I_I_FC_O1_NEG
ST   AXLSREF81.x_MIN_LS                             * Min Limit switch

LD   I_I_FC_O1_POS
ST   AXLSREF81.x_MAX_LS                             * Max Limit switch

LD   ALWAYS_ZERO
ST   AXLSREF81.x_REF_S                              * Reference switch

CAL  AXLSREF81

LD   AXLSREF81.y_MIN_LS                             * Min Limit switch
ST   GESTAX81.xMinusLS                              * Negative limit switch

LD   AXLSREF81.y_MAX_LS                             * Max Limit switch
ST   GESTAX81.xPlusLS                               * Positive limit switch

LD   AXLSREF81.y_REF_S                              * Reference switch
ST   GESTAX81.xRefLS                                * Reference
***

LD   MainAxesPowerAllowed
AND  MainAxesPower                                  * PON
ST   GESTAX81.xCloseLoop

LD   Sel_Y_Ch9
ST   GESTAX81.xSelected

***************************************
* Change REF quota for ABS reference
***************************************
CAL  RTRIG_AX_SEL81(CLK:=GESTAX81.xSelected)

LD   RTRIG_AX_SEL81.Q
JMPCN NoSel81
LD   ActualQtaAbsRef                                ** Absolute homing quota
ST   QtaRefAbsSet                                   ** Absolute homing quota setting
NoSel81:

LD   GESTAX81.xSelected
AND  %nvel14.0                                      * Se Vale 1 ?gestito "Encoder Assoluto" (Da Configura Asse)
AND (
LD   ActualQtaAbsRef                                ** Absolute homing quota
NE   QtaRefAbsSet                                   ** Absolute homing quota setting
)
JMPCN NoEq81

LD   QtaRefAbsSet                                   ** Absolute homing quota setting
ST   ActualQtaAbsRef                                ** Absolute homing quota
NoEq81:
***************************************

LD   Pul_Jogp                                       ** (gPlc0.4)jog+ pushbutton
AND  GESTAX81.xSelected
ANDN PlcEmerGen                                     ** M0.10 Emergenza generale
AND  GESTAX81.xCloseLoop
ST   GESTAX81.xJogPlus

LD   Pul_Jogm                                       ** (gPlc0.5)jog- pushbutton
AND  GESTAX81.xSelected
ANDN PlcEmerGen                                     ** M0.10 Emergenza generale
AND  GESTAX81.xCloseLoop
*ANDN CMD_HOLDMOVING_CH9.1
ST   GESTAX81.xJogMinus

LD   %nvel14.0                                      * Se Vale 1 ?gestito "Encoder Assoluto" (Da Configura Asse)
ST   GESTAX81.xZeroForced                           * Forzamento asse tarato

LD   GESTAX2_xHoldMoving                            * Richiesta blocco avanzamento
OR(
LD   CMD_HOLDMOVING_CH9.1                           ** M203 Hold moving command axis CH5 (bit0=X, bit1=Y...)
*AND  UnSupp_81_GoUp
)
ST   GESTAX81.xHoldMoving                           * Richiesta blocco avanzamento

LD   Res_Axes                                       ** (gPlc25.1) reset axes disable electric shaft
ST   GESTAX81.xUnlock

LDN  ch9_in_ref                                     ** channel 3 in ref
ST   GESTAX81.xEnFIR                                * Abilita filtri FIR
ST   GESTAX81.xEnFrComp                             ** Abilita friction compensation

LD   ALWAYS_ZERO                                    ** PLCFLAGS.0  Flag sempre stato off
ST   GESTAX81.xDisLimiter

LD   %cn0.rc8.3                                     * ch0 in alarm
OR   %cn3.rc8.3                                     * ch3 in alarm
**OR   EmerINC
ST   GESTAX81.xSetAlarm                             ** Forzamento allarme asse

LD   usrReqGrantSupLat1
ST   GESTAX81.xFromPlc

CAL  GESTAX81

LD   GESTAX81.yDriveNotEn
S    %PLCerr3.24

LD   BSG_INC                                        ** rg1.2 Selezione modo INC (inc.fissi)
JMPCN SVIX81

LD   %pa59                                          * Velocit?di Repos
MUL  1000
DIV  60
MUL  MainChFeedrate                                 ** (gPlc16) feed degli assi (%)
DIV  100
ST   %ra50                                          * Limitazione velocita' massima interpolazione

SVIX81:
NOAX81:

********************************************************************************
* Unload Support 1 (ax71)
********************************************************************************
PATH %ax82
PATH %ax_lsref82

***************************************
*   POWER ON (PON)
***************************************
LD   %pa3.31            * Simulato
ORN  %cc1.2             * Maschera assi associata al canale
OR(
LD   %nvel11            ** 3,4=CANopen, Ecat
EQ   3
)
OR(
LD   %nvel11            ** 3,4=CANopen, Ecat
EQ   4
)
ST   Pon_UnSupp_82      ** PON unload support axis
***************************************

LDN  %ra3.2                                         * ra3.2  Direzione moto asse avanti
OR   %ra0.9                                         * ra0.9 Comando indietro
AND  %ra3.13                                        * ra3.13  Ordine di moto
ST   UnSupp_82_GoUp

LD  %cc1.2           * Maschera assi associata al canale 8
JMPCN NOAX82

***
*   LIMIT SWITCH & REFERENCE SWITCH

LD   %lsrefmode
ST   AXLSREF82.x_REF_mode        * 0=use ref switch...

LD   %lsreflevel
ST   AXLSREF82.x_TYPE_LS         * (1=NC, 0=NO)

LD   I_I_FC_O2_NEG
ST   AXLSREF82.x_MIN_LS          * Min Limit switch

LD   I_I_FC_O2_POS
ST   AXLSREF82.x_MAX_LS          * Max Limit switch

LD   ALWAYS_ZERO
ST   AXLSREF82.x_REF_S           * Reference switch

CAL  AXLSREF82

LD   AXLSREF82.y_MIN_LS          * Min Limit switch
ST   GESTAX82.xMinusLS           * Negative limit switch

LD   AXLSREF82.y_MAX_LS          * Max Limit switch
ST   GESTAX82.xPlusLS            * Positive limit switch

LD   AXLSREF82.y_REF_S           * Reference switch
ST   GESTAX82.xRefLS             * Reference
***

LD   MainAxesPowerAllowed
AND  MainAxesPower               * PON
ST   GESTAX82.xCloseLoop

LD   Sel_Z_Ch9
ST   GESTAX82.xSelected

***************************************
* Change REF quota for ABS reference
***************************************
CAL  RTRIG_AX_SEL82(CLK:=GESTAX82.xSelected)

LD   RTRIG_AX_SEL82.Q
JMPCN NoSel72
LD   ActualQtaAbsRef               ** Absolute homing quota
ST   QtaRefAbsSet                  ** Absolute homing quota setting
NoSel72:

LD   GESTAX82.xSelected
AND  %nvel14.0                     * Se Vale 1 � gestito "Encoder Assoluto" (Da Configura Asse)
AND (
LD   ActualQtaAbsRef               ** Absolute homing quota
NE   QtaRefAbsSet                  ** Absolute homing quota setting
)
JMPCN NoEq82

LD   QtaRefAbsSet                  ** Absolute homing quota setting
ST   ActualQtaAbsRef               ** Absolute homing quota
NoEq82:
***************************************

LD   Pul_Jogp                      ** (gPlc0.4)jog+ pushbutton
AND  GESTAX82.xSelected
ANDN PlcEmerGen                      ** M0.10 Emergenza generale
AND  GESTAX82.xCloseLoop
ST   GESTAX82.xJogPlus

LD   Pul_Jogm                      ** (gPlc0.5)jog- pushbutton
AND  GESTAX82.xSelected
ANDN PlcEmerGen                      ** M0.10 Emergenza generale
AND  GESTAX82.xCloseLoop
*ANDN CMD_HOLDMOVING_CH9.2
ST   GESTAX82.xJogMinus

LD   %nvel14.0                     * Se Vale 1 � gestito "Encoder Assoluto" (Da Configura Asse)
ST   GESTAX82.xZeroForced          * Forzamento asse tarato

LD   GESTAX2_xHoldMoving           * Richiesta blocco avanzamento
OR(
LD   CMD_HOLDMOVING_CH9.2          ** M203 Hold moving command axis CH5 (bit0=X, bit1=Y...)
*AND  UnSupp_82_GoUp
)
ST   GESTAX82.xHoldMoving          * Richiesta blocco avanzamento

LD   Res_Axes                      ** (gPlc25.1) reset axes disable electric shaft
ST   GESTAX82.xUnlock

LDN  ch9_in_ref                    ** channel 3 in ref
ST   GESTAX82.xEnFIR               * Abilita filtri FIR
ST   GESTAX82.xEnFrComp            ** Abilita friction compensation

LD   ALWAYS_ZERO                   ** PLCFLAGS.0  Flag sempre stato off
ST   GESTAX82.xDisLimiter

LD   %cn0.rc8.3                    * ch0 in alarm
OR   %cn3.rc8.3                    * ch3 in alarm
**OR   EmerINC
ST   GESTAX82.xSetAlarm            ** Forzamento allarme asse

LD   usrReqGrantSupLat2
ST   GESTAX82.xFromPlc

CAL  GESTAX82

LD   GESTAX82.yDriveNotEn
S    %PLCerr3.25

LD   BSG_INC                       ** rg1.2 Selezione modo INC (inc.fissi)
JMPCN SVIX82

LD   %pa59                         * Velocit� di Repos
MUL  1000
DIV  60
MUL  MainChFeedrate                ** (gPlc16) feed degli assi (%)
DIV  100
ST   %ra50                         * Limitazione velocita' massima interpolazione

SVIX82:
NOAX82:

********************************************************************************
* Unload Support 2 (ax73)
********************************************************************************
PATH %ax83
PATH %ax_lsref83

***************************************
*   POWER ON (PON)
***************************************
LD   %pa3.31                                        * Simulato
ORN  %cc1.3                                         * Maschera assi associata al canale
OR(
LD   %nvel11                                        ** 3,4=CANopen, Ecat
EQ   3
)
OR(
LD   %nvel11                                        ** 3,4=CANopen, Ecat
EQ   4
)
ST   Pon_UnSupp_83                                  ** PON unload support axis
***************************************

LDN  %ra3.2                                         * ra3.2  Direzione moto asse avanti
OR   %ra0.9                                         * ra0.9 Comando indietro
AND  %ra3.13                                        * ra3.13  Ordine di moto
ST   UnSupp_83_GoUp

LD  %cc1.3                                          * Maschera assi associata al canale 8
JMPCN NOAX83

***
*   LIMIT SWITCH & REFERENCE SWITCH

LD   %lsrefmode
ST   AXLSREF83.x_REF_mode                           * 0=use ref switch...

LD   %lsreflevel
ST   AXLSREF83.x_TYPE_LS                            * (1=NC, 0=NO)

LD   I_I_FC_O3_NEG
ST   AXLSREF83.x_MIN_LS                             * Min Limit switch

LD   I_I_FC_O3_POS
ST   AXLSREF83.x_MAX_LS                             * Max Limit switch

LD   ALWAYS_ZERO
ST   AXLSREF83.x_REF_S                              * Reference switch

CAL  AXLSREF83

LD   AXLSREF83.y_MIN_LS                             * Min Limit switch
ST   GESTAX83.xMinusLS                              * Negative limit switch

LD   AXLSREF83.y_MAX_LS                             * Max Limit switch
ST   GESTAX83.xPlusLS                               * Positive limit switch

LD   AXLSREF83.y_REF_S                              * Reference switch
ST   GESTAX83.xRefLS                                * Reference
***

LD   MainAxesPowerAllowed
AND  MainAxesPower                                  * PON
ST   GESTAX83.xCloseLoop

LD   Sel_U_Ch9
ST   GESTAX83.xSelected

***************************************
* Change REF quota for ABS reference
***************************************
CAL  RTRIG_AX_SEL83(CLK:=GESTAX83.xSelected)

LD   RTRIG_AX_SEL83.Q
JMPCN NoSel83
LD   ActualQtaAbsRef                                ** Absolute homing quota
ST   QtaRefAbsSet                                   ** Absolute homing quota setting
NoSel83:

LD   GESTAX83.xSelected
AND  %nvel14.0                                      * Se Vale 1 ?gestito "Encoder Assoluto" (Da Configura Asse)
AND (
LD   ActualQtaAbsRef                                ** Absolute homing quota
NE   QtaRefAbsSet                                   ** Absolute homing quota setting
)
JMPCN NoEq83

LD   QtaRefAbsSet                                   ** Absolute homing quota setting
ST   ActualQtaAbsRef                                ** Absolute homing quota
NoEq83:
***************************************

LD   Pul_Jogp                                       ** (gPlc0.4)jog+ pushbutton
AND  GESTAX83.xSelected
ANDN PlcEmerGen                                     ** M0.10 Emergenza generale
AND  GESTAX83.xCloseLoop
ST   GESTAX83.xJogPlus

LD   Pul_Jogm                                       ** (gPlc0.5)jog- pushbutton
AND  GESTAX83.xSelected
ANDN PlcEmerGen                                     ** M0.10 Emergenza generale
AND  GESTAX83.xCloseLoop
*ANDN CMD_HOLDMOVING_CH9.3
ST   GESTAX83.xJogMinus

LD   %nvel14.0                                      * Se Vale 1 ?gestito "Encoder Assoluto" (Da Configura Asse)
ST   GESTAX83.xZeroForced                           * Forzamento asse tarato

LD   GESTAX2_xHoldMoving                            * Richiesta blocco avanzamento
OR(
LD   CMD_HOLDMOVING_CH9.3                           ** M203 Hold moving command axis CH5 (bit0=X, bit1=Y...)
*AND  UnSupp_83_GoUp
)
ST   GESTAX83.xHoldMoving                           * Richiesta blocco avanzamento

LD   Res_Axes                                       ** (gPlc25.1) reset axes disable electric shaft
ST   GESTAX83.xUnlock

LDN  ch9_in_ref                                     ** channel 3 in ref
ST   GESTAX83.xEnFIR                                * Abilita filtri FIR
ST   GESTAX83.xEnFrComp                             ** Abilita friction compensation

LD   ALWAYS_ZERO                                    ** PLCFLAGS.0  Flag sempre stato off
ST   GESTAX83.xDisLimiter

LD   %cn0.rc8.3                                     * ch0 in alarm
OR   %cn3.rc8.3                                     * ch3 in alarm
**OR   EmerINC
ST   GESTAX83.xSetAlarm                             ** Forzamento allarme asse

LD   usrReqGrantSupLat3
ST   GESTAX83.xFromPlc

CAL  GESTAX83

LD   GESTAX83.yDriveNotEn
S    %PLCerr3.26

LD   BSG_INC                                        ** rg1.2 Selezione modo INC (inc.fissi)
JMPCN SVIX83

LD   %pa59                                          * Velocit?di Repos
MUL  1000
DIV  60
MUL  MainChFeedrate                                 ** (gPlc16) feed degli assi (%)
DIV  100
ST   %ra50                                          * Limitazione velocita' massima interpolazione

SVIX83:
NOAX83:

********************************************************************************
* Unload Support 3 (ax74)
********************************************************************************
PATH %ax84
PATH %ax_lsref84

***************************************
*   POWER ON (PON)
***************************************
LD   %pa3.31                                        * Simulato
ORN  %cc1.4                                         * Maschera assi associata al canale
OR(
LD   %nvel11                                        ** 3,4=CANopen, Ecat
EQ   3
)
OR(
LD   %nvel11                                        ** 3,4=CANopen, Ecat
EQ   4
)
ST   Pon_UnSupp_84                                  ** PON unload support axis
***************************************

LDN  %ra3.2                                         * ra3.2  Direzione moto asse avanti
OR   %ra0.9                                         * ra0.9 Comando indietro
AND  %ra3.13                                        * ra3.13  Ordine di moto
ST   UnSupp_84_GoUp

LD  %cc1.4                                          * Maschera assi associata al canale 8
JMPCN NOAX84

***
*   LIMIT SWITCH & REFERENCE SWITCH

LD   %lsrefmode
ST   AXLSREF84.x_REF_mode                           * 0=use ref switch...

LD   %lsreflevel
ST   AXLSREF84.x_TYPE_LS                            * (1=NC, 0=NO)

LD   I_I_FC_O4_NEG
ST   AXLSREF84.x_MIN_LS                             * Min Limit switch

LD   I_I_FC_O4_POS
ST   AXLSREF84.x_MAX_LS                             * Max Limit switch

LD   ALWAYS_ZERO
ST   AXLSREF84.x_REF_S                              * Reference switch

CAL  AXLSREF84

LD   AXLSREF84.y_MIN_LS                             * Min Limit switch
ST   GESTAX84.xMinusLS                              * Negative limit switch

LD   AXLSREF84.y_MAX_LS                             * Max Limit switch
ST   GESTAX84.xPlusLS                               * Positive limit switch

LD   AXLSREF84.y_REF_S                              * Reference switch
ST   GESTAX84.xRefLS                                * Reference
***

LD   MainAxesPowerAllowed
AND  MainAxesPower                                  * PON
ST   GESTAX84.xCloseLoop

LD   Sel_V_Ch9
ST   GESTAX84.xSelected

***************************************
* Change REF quota for ABS reference
***************************************
CAL  RTRIG_AX_SEL84(CLK:=GESTAX84.xSelected)

LD   RTRIG_AX_SEL84.Q
JMPCN NoSel84
LD   ActualQtaAbsRef                                ** Absolute homing quota
ST   QtaRefAbsSet                                   ** Absolute homing quota setting
NoSel84:

LD   GESTAX84.xSelected
AND  %nvel14.0                                      * Se Vale 1 ?gestito "Encoder Assoluto" (Da Configura Asse)
AND (
LD   ActualQtaAbsRef                                ** Absolute homing quota
NE   QtaRefAbsSet                                   ** Absolute homing quota setting
)
JMPCN NoEq84

LD   QtaRefAbsSet                                   ** Absolute homing quota setting
ST   ActualQtaAbsRef                                ** Absolute homing quota
NoEq84:
***************************************

LD   Pul_Jogp                                       ** (gPlc0.4)jog+ pushbutton
AND  GESTAX84.xSelected
ANDN PlcEmerGen                                     ** M0.10 Emergenza generale
AND  GESTAX84.xCloseLoop
ST   GESTAX84.xJogPlus

LD   Pul_Jogm                                       ** (gPlc0.5)jog- pushbutton
AND  GESTAX84.xSelected
ANDN PlcEmerGen                                     ** M0.10 Emergenza generale
AND  GESTAX84.xCloseLoop
*ANDN CMD_HOLDMOVING_CH9.4
ST   GESTAX84.xJogMinus

LD   %nvel14.0                                      * Se Vale 1 ?gestito "Encoder Assoluto" (Da Configura Asse)
ST   GESTAX84.xZeroForced                           * Forzamento asse tarato

LD   GESTAX2_xHoldMoving                            * Richiesta blocco avanzamento
OR(
LD   CMD_HOLDMOVING_CH9.4                           ** M203 Hold moving command axis CH5 (bit0=X, bit1=Y...)
*AND  UnSupp_84_GoUp
)
ST   GESTAX84.xHoldMoving                           * Richiesta blocco avanzamento

LD   Res_Axes                                       ** (gPlc25.1) reset axes disable electric shaft
ST   GESTAX84.xUnlock

LDN  ch9_in_ref                                     ** channel 3 in ref
ST   GESTAX84.xEnFIR                                * Abilita filtri FIR
ST   GESTAX84.xEnFrComp                             ** Abilita friction compensation

LD   ALWAYS_ZERO                                    ** PLCFLAGS.0  Flag sempre stato off
ST   GESTAX84.xDisLimiter

LD   %cn0.rc8.3                                     * ch0 in alarm
OR   %cn3.rc8.3                                     * ch3 in alarm
**OR   EmerINC
ST   GESTAX84.xSetAlarm                             ** Forzamento allarme asse

LD   usrReqGrantSupLat4
ST   GESTAX84.xFromPlc

CAL  GESTAX84

LD   GESTAX84.yDriveNotEn
S    %PLCerr3.27

LD   BSG_INC                                        ** rg1.2 Selezione modo INC (inc.fissi)
JMPCN SVIX84

LD   %pa59                                          * Velocit?di Repos
MUL  1000
DIV  60
MUL  MainChFeedrate                                 ** (gPlc16) feed degli assi (%)
DIV  100
ST   %ra50                                          * Limitazione velocita' massima interpolazione

SVIX84:
NOAX84:

**************************
* Acknowledg funzioni "M"
**************************
*
LD   %PLCFLAGS.0
ST   CH9END.xWaitMFun

CAL  CH9END

END_FUNCTION

(* ---- usrCmd.plc ---- *)
*******************************************************************************
*   usrCnd.plc
*   ESAutomotion
*   LASER machine
*******************************************************************************
VAR_IN_OUT
#include "mem.inc"
#include "usrIol.inc"
END_VAR
#include "usrMem.inc"

FUNCTION COMMAND_TO_MAIN

*CH3
* Hold V axis

LD   Hold_U_Z1Supp
OR   Hold_U_Z2Supp
OR   Hold_U_Z3Supp
OR   Hold_U_Z4Supp
OR   Hold_U_Z5Supp
OR   Hold_U_SupUnHorAx85
OR   Hold_U_SupUnHorAx86
OR   Hold_U_SupUnHorAx87
OR   Hold_U_SupUnHorAx88
OR   M_HoldAx_V
ST   CMD_HOLDMOVING_CH3.4            ** M202 Hold moving command axis CH3 (bit0=X, bit1=Y...)

* Hold X-U
LD   Hold_U_Z1SuppLoad
OR   Hold_U_Z2SuppLoad
OR   Hold_U_Z3SuppLoad
OR   Hold_U_Z4SuppLoad
OR   HoldO1Ax30_HOR
OR   HoldO2Ax30_HOR
OR   HoldO3Ax30_HOR
OR   HoldO4Ax30_HOR
OR   %PLCmsg8.5
OR   M_HoldAx_U
ST   CMD_HOLDMOVING_CH3.0            ** M202 Hold moving command axis CH3 (bit0=X, bit1=Y...)

* CH8 (Unloader)

LD   HoldZ1Supp
ST   CMD_HOLDMOVING_CH8.1            ** M203 Hold moving command axis CH5 (bit0=X, bit1=Y...)

LD   HoldZ2Supp
ST   CMD_HOLDMOVING_CH8.2            ** M203 Hold moving command axis CH5 (bit0=X, bit1=Y...)

LD   HoldZ3Supp
ST   CMD_HOLDMOVING_CH8.3            ** M203 Hold moving command axis CH5 (bit0=X, bit1=Y...)

LD   HoldZ4Supp
ST   CMD_HOLDMOVING_CH8.4            ** M203 Hold moving command axis CH5 (bit0=X, bit1=Y...)

LD   HoldZ5Supp
ST   CMD_HOLDMOVING_CH8.5            ** M203 Hold moving command axis CH5 (bit0=X, bit1=Y...)

* CH5

* Grant Request

LD   usrReqGrantSupL1
ST   GRANT5.1

LD   usrReqGrantSupL2
ST   GRANT5.2

LD   usrReqGrantSupL3
ST   GRANT5.3

LD   usrReqGrantSupL4
ST   GRANT5.4

* Hold support axes

LD   HoldZ1SuppLoad
ST   CMD_HOLDMOVING_CH5.1

LD   HoldZ2SuppLoad
ST   CMD_HOLDMOVING_CH5.2

LD   HoldZ3SuppLoad
ST   CMD_HOLDMOVING_CH5.3

LD   HoldZ4SuppLoad
ST   CMD_HOLDMOVING_CH5.4

* Hold support Lateral axes

LD   HoldO1SuppLoad_LAT
ST   CMD_HOLDMOVING_CH9.1

LD   HoldO2SuppLoad_LAT
ST   CMD_HOLDMOVING_CH9.2

LD   HoldO3SuppLoad_LAT
ST   CMD_HOLDMOVING_CH9.3

LD   HoldO4SuppLoad_LAT
ST   CMD_HOLDMOVING_CH9.4

*
END_FUNCTION

(* ---- usrGen.plc ---- *)
#include "iol.inc"
#include "usrMem.inc"

VAR
TON36:                TON;
appoggio:             BOOL;
State_AutOrg:         BOOL;
CurrState:            DWORD;
DangerThresld:        DWORD;
YZatParking:          DWORD;
emercaseA:            DWORD;
emercaseB:            DWORD;
R_TRIG_M3:            R_TRIG;
R_TRIG_Heading:       R_TRIG;
F_TRIG_Heading:       F_TRIG;
END_VAR

VAR_IN_OUT
#include "usrIol.inc"
END_VAR

FUNCTION M_WAIT

LD   FS_WaitM
OR   MS_WaitM
OR   (
LD   Fun_M730_Ch0
ANDN I_I_Loader_Reach_Pos
)
OR   (
LD   Fun_M731_Ch0
ANDN I_I_Loader_Back_Pos
)
*OR   WaitLoadM
*LD   WaitServiceCH7
*OR   WaitServiceCH8
*OR   WaitServiceCH9
ST   WaitMfunc0Usr                 ** wait m function on ch0

*//============================================================================
*// Heading Function Origin Acquiring Management
*// - HMI Heading Require Enable Management
*//============================================================================
CAL  R_TRIG_Heading(CLK=%LSRPlcOp0.21)
LD   R_TRIG_Heading.Q
ANDN %cn0.rc8.0
JMPCN REC_STATUS
LD   OriginAtStar
ST   State_AutOrg
REC_STATUS:

LD   %LSRPlcOp0.21
JMPCN FORCE_EN_ORG
LD   %PLCFLAGS.1
ST   OriginAtStar
FORCE_EN_ORG:

LD   R_TRIG_Heading.Q
ANDN %cn0.rc8.0
ANDN State_AutOrg
S    OriginAtStar

CAL  F_TRIG_Heading(CLK=%LSRPlcOp0.21)
LD   F_TRIG_Heading.Q
ANDN %cn0.rc8.0
ANDN State_AutOrg
R    OriginAtStar

*//============================================================================
*// Startup Machine with 3D viewer
*//============================================================================
LD   %PLCFLAGS.8
R    guiShowISO

*//============================================================================
*// WeldSeam Detection
*//============================================================================
LD   visCameraPiston
AND  %cn0.rc8.0
OR   Btn_Weld_Piston           * Toggle
ST   O_O_Detec_Weld_Piston

LD   %cn0.rc8.0
AND  Btn_Weld_Piston
R    Btn_Weld_Piston

LD   IsoCameraToDetec
AND  %cn0.rc8.0
OR   Btn_Weld_En               * Pulses
ST   O_O_Detec_Weld

LDN  %cn0.rc8.0
JMPCN CLRSTATUS
     LD   0
	 ST   O_O_WeldDetec_En
     ST   IsoCameraToDetec
	 ST   visCameraPiston
	 ST   CN3_REQ_VYZ_ISO
CLRSTATUS:

*//============================================================================
*// Following supports quote monitoring
*//============================================================================
LD   %ax50.ra4
SUB  2000           *2mm
ST   DangerThresld

LD   EnWriteBlendSwitch
OR   EnWriteBlendSwitch1
AND  %cn0.rc8.0
JMPCN INSIDETUB
     LD   %ax51.ra4
     LT   DangerThresld
     AND  %cn5.cc1.1
     OR(
	 LD   %ax52.ra4
     LT   DangerThresld
     AND  %cn5.cc1.2
	 )
     OR(
	 LD   %ax53.ra4
     LT   DangerThresld
     AND  %cn5.cc1.3
	 )
     OR(
	 LD   %ax54.ra4
     LT   DangerThresld
     AND  %cn5.cc1.4
	 )
	 * Unloader
	 OR(
	 LD   %ax72.ra4
	 LT   DangerThresld
	 AND  %cn8.cc1.2
	 )
	 OR(
	 LD   %ax71.ra4
	 LT   DangerThresld
	 AND  %cn8.cc1.1
	 )
     OR(
	 LD   %ax73.ra4
	 LT   DangerThresld
	 AND  %cn8.cc1.3
	 )
	 OR(
	 LD   %ax74.ra4
	 LT   DangerThresld
	 AND  %cn8.cc1.4
	 )
	 OR(
	 LD   %ax75.ra4
	 LT   DangerThresld
	 AND  %cn8.cc1.5
	 )
	 ST   Emer_Sup_QtaErr

	 LD   Emer_Sup_QtaErr
	 S    %PLCerr20.24

INSIDETUB:

LDN  %cn0.rc8.0
OR   Pul_Reset
R    %PLCerr20.24
R    iso_G510_StartDM4
R    %PLCmsg0.8

*//============================================================================
*// Spindle Quote monitoring (gearing software limit protection) - 3mm
*// - to ensure safety in case of cad-cam mistake
*//============================================================================
LD   GESTAX36_xHoldMoving
ANDN %ax36.ra3.0
AND  %cn3.cc1.5
ST   appoggio
CAL  TON36(IN=appoggio,PT=1000)

LD   %ax30.ra4
SUB  3000
GT   %ax30.pa22
OR(
LD   %ax30.ra4
ADD  3000
LT   %ax30.pa21
)
OR(
LD   %ax36.ra4
SUB  3000
GT   %ax36.pa22
AND  %cn3.cc1.5
)
OR(
LD   %ax36.ra4
ADD  3000
LT   %ax36.pa21
AND  %cn3.cc1.5
)
OR(
LD   %ax31.ra4
SUB  3000
GT   %ax31.pa22
AND  %cn3.cc1.4
)
OR(
LD   %ax31.ra4
ADD  3000
LT   %ax31.pa21
AND  %cn3.cc1.4
)
OR   TON36.Q
AND  %cn0.rc8.0
ANDN ch0_in_ref
ANDN ch0_in_jog
S    %PLCerr20.25

LD   Pul_Reset
R    %PLCerr20.25

*//============================================================================
*// B Bevel and W Middle Spindle Management
*// - when W not at limit not able to move B manaully
*// - W anticolision condition to check with B angle
*//============================================================================
LD   %ax29.pa22
SUB  %ax29.ra4
ABS
LT   20000
AND   (
LD   %ax28.pa21
SUB  %ax28.ra4
ABS
LT   20000
)
ST   YZatParking

LD   45000
SIN
MULDIV(M=%twi1.htwi.oarh.dZ,D=1000)
ADD  10000
ST   tmp_lim_holder

LD   %ax36.pa22
SUB  tmp_lim_holder
ST   safedisPosQta

LD   %ax36.pa21
ADD  tmp_lim_holder
ST   safedisNegQta

*LD   Gest5Ax
*AND  %cn3.cc1.5
*JMPCN STATUSONLYBVL

* Jog Mode to hold ****************************************** //

	 LD   %ax36.ra92
	 SUB (
	 LD   %ax33.ra92
	 SIN
	 MULDIV(M=%twi1.htwi.oarh.dZ,D=1000)
     )
	 LT   safedisPosQta
	 AND(
	 LD   %ax33.ra4
	 GE   0
	 )
	 OR(
	      LD   %ax36.ra92
		  LT   safedisPosQta
	 )
	 AND(
	 LD   %ax36.ra4
	 GE   0
	 )
	 ANDN YZatParking
	 ANDN ch0_in_ref
	 ANDN %cn0.rc8.0
	 ST   %PLCmsg8.9   * Stop W-, B+

	 LD   %ax36.ra92
	 SUB (
	 LD   %ax33.ra92
	 SIN
	 MULDIV(M=%twi1.htwi.oarh.dZ,D=1000)
     )
	 GT   safedisNegQta
	 AND(
	 LD   %ax33.ra4
	 LT   0
	 )
	 OR(
	      LD   %ax36.ra92
		  GT   safedisNegQta
	 )
	 AND(
	 LD   %ax36.ra4
	 LT   0
	 )
	 ANDN YZatParking
	 ANDN ch0_in_ref
	 ANDN %cn0.rc8.0
	 ST   %PLCmsg8.10  * Stop W+, B-

* Aut Mode to Emer (3mm more) ******************************* //

	 LD   %ax36.ra4
	 SUB (
	 LD   %ax33.ra4
	 SIN
	 MULDIV(M=%twi1.htwi.oarh.dZ,D=1000)
     )
	 ST   dynamicBsafe

	 LD   dynamicBsafe
	 ADD  3000
	 LT   safedisPosQta
	 AND(
	 LD   %ax33.ra4
	 GE   0
	 )
	 OR(
	      LD   %ax36.ra4
		  ADD  3000
		  LT   safedisPosQta
	 )
	 AND(
	 LD   %ax36.ra4
	 GE   0
	 )
	 ANDN YZatParking
	 ANDN ch0_in_ref
	 ST   emercaseA

	 LD   dynamicBsafe
	 SUB  3000
	 GT   safedisNegQta
	 AND(
	 LD   %ax33.ra4
	 LT   0
	 )
	 OR(
	      LD   %ax36.ra4
		  SUB  3000
		  GT   safedisNegQta
	 )
	 AND(
	 LD   %ax36.ra4
	 LT   0
	 )
	 ANDN YZatParking
	 ANDN ch0_in_ref
	 ST   emercaseB

	 LD   emercaseA
	 OR   emercaseB
     AND  %cn0.rc8.0
	 S    %PLCerr20.26  * Anticolision between B and W

     LD   %ax29.ra0.9   * Z-
     OR   %ax28.ra0.8   * Y+
     OR   %ax36.ra0.9   * W-
     AND(
     LD   safedisPosQta
     SUB  %ax36.ra4
     GT   5000
     )
	 AND(
	 LD   %ax36.ra4
	 GE   0
	 )
     OR  (
          LD   %ax29.ra0.9  * Z-
          OR   %ax28.ra0.8  * Y+
          OR   %ax36.ra0.8  * W+
          AND(
          LD   %ax36.ra4
          SUB  safedisNegQta
          GT   5000
          )
		  AND(
	      LD   %ax36.ra4
	      LT   0
	      )
     )
     ANDN YZatParking
     ANDN ch0_in_ref
     S    %PLCerr20.22  * Anticolision between Z and W

	 LD   Pul_Reset
     R    %PLCerr20.22
     R    %PLCerr20.26

STATUSONLYBVL:

*//============================================================================
*// Real Tube Position Update
*//============================================================================
PATH %funz[19]

LD   iso_G510_StartDM4
OR(
LDN  O_O_Mobile_Spindle_Slave_Close
AND  iso_G520_Running
)
JMPC FREEZEUPDATE

LD   O_O_Mobile_Spindle_Close
ANDN O_O_Mobile_Spindle_Slave_Close
JMPCN STATEM2
     LD  2
	 ST  CurrState
STATEM2:

LD   O_O_Mobile_Spindle_Close
AND  O_O_Mobile_Spindle_Slave_Close
JMPCN STATEM3
     LD  3
	 ST  CurrState
STATEM3:

LDN  O_O_Mobile_Spindle_Close
AND  O_O_Mobile_Spindle_Slave_Close
JMPCN STATEM3M4
     LD  4
	 ST  CurrState
STATEM3M4:

LD   CurrState
EQ   3
ST   appoggio
CAL  R_TRIG_M3(CLK=appoggio)
LD   R_TRIG_M3.Q
JMPCN RECORDLEN
     LD   %ax31.ra24
     SUB  %ax30.ra24
	 ABS
     ST   OFFSETM4
RECORDLEN:

LD   CurrState
EQ   4
JMPCN MASTERM4P
	 LD   %ax0.ra24
	 SUB  %ax31.ra24
	 SUB  OFFSETM4
	 ADD  ORIGPRGX
     ST   tmpartOffset
MASTERM4P:

LD   CurrState
EQ   2
OR(
LD   CurrState
EQ   3
)
JMPCN MASTERM2P
     LD   CurrState
     EQ   2
	 JMPCN CLRM2ZERO
          LD   0
	      ST   OFFSETM4
     CLRM2ZERO:

	 LD   %ax0.ra24
	 SUB  %ax30.ra24
     ADD  ORIGPRGX
     ST   tmpartOffset
MASTERM2P:

FREEZEUPDATE:

*//============================================================================

END_FUNCTION

(* ---- usrIOCon.plc ---- *)
#include "iol.inc"
#include "usrMem.inc"

VAR
#include "Iof.inc"
#include "usrIof.inc"

Appoggio:                   BOOL;
Ton_PrgRun:                 TON;
TON_SpindleFix_Close_C1:    TON; *YANG230905
TON_SpindleFix_Open_C1:     TON;
TON_Spindle_Slave_Open_C2:  TON;
TON_Spindle_Slave_Close_C2: TON;
FTRIG_EMER:                 F_TRIG;
END_VAR

VAR_IN_OUT
#include "usrIol.inc"
#include "mem.inc"
END_VAR

*******************************************************
* USER INPUT CONFIGURATION
*******************************************************

FUNCTION USR_INP_CONFIG

LDN  I_TubeMobile_Spindle
ST   I_I_TubeMobile_Spindle

LDN  I_TubeFix_Spindle
ST   I_I_TubeFix_Spindle

LD   I_Pul_Mobile_Spindle_Close
ST   I_I_Pul_Mobile_Spindle_Close
ST   %PLCmsg8.7

LD   I_Pul_Mobile_Spindle_Open
ST   I_I_Pul_Mobile_Spindle_Open
ST   %PLCmsg8.6

*LD   I_Mobile_Spindle_Open
LD   O_Mobile_Spindle_Open
ST   I_I_Mobile_Spindle_Open

*LD   I_Mobile_Spindle_Close
LD   O_Mobile_Spindle_Close
ST   I_I_Mobile_Spindle_Close

*LD   I_Mobile_Spindle_Slave_Open
LD   O_Mobile_Spindle_Slave_Open
ST   I_I_Mobile_Spindle_Slave_Open

*LD   I_Mobile_Spindle_Slave_Close
LD   O_Mobile_Spindle_Slave_Close
ST   I_I_Mobile_Spindle_Slave_Close

*LD   I_FixedSpindle_Open                     ** yang no sensor in GWK 230907
LD   O_O_SpindleFix_Open
ST   I_I_FixedSpindle_Open

*LD   I_FixedSpindle_Close                    ** yang no sensor in GWK 230907
LD   O_O_SpindleFix_Close
ST   I_I_FixedSpindle_Close

LD   I_Butt_Open_Mobile
ST   I_I_Butt_Open_Mobile

LD   I_Butt_Close_Mobile
ST   I_I_Butt_Close_Mobile

LD   I_Butt_Open_Fix
ST   I_I_Butt_Open_Fix

LD   I_Butt_Close_Fix
ST   I_I_Butt_Close_Fix

LD    I_Support_1_Dwn
ST   I_I_Support_1_Dwn

LD    I_Support_2_Dwn
ST   I_I_Support_2_Dwn

LD    I_Support_3_Dwn
ST   I_I_Support_3_Dwn

LD    I_Support_4_Dwn
ST   I_I_Support_4_Dwn

LDN   I_Support_5_Dwn
ST   I_I_Support_5_Dwn

LDN   I_Support_6_Dwn
ST   I_I_Support_6_Dwn

LDN   I_Support_7_Dwn
ST   I_I_Support_7_Dwn

LD   I_Support_1_Dwn_Un
ST   I_I_Support_1_Dwn_Un

LD   I_Support_2_Dwn_Un
ST   I_I_Support_2_Dwn_Un

LD   I_Support_3_Dwn_Un
ST   I_I_Support_3_Dwn_Un

LD   I_Support_4_Dwn_Un
ST   I_I_Support_4_Dwn_Un

LD   I_Support_5_Dwn_Un
ST   I_I_Support_5_Dwn_Un

LD   I_Support_6_Dwn_Un
ST   I_I_Support_6_Dwn_Un

LD   I_Support_7_Dwn_Un
ST   I_I_Support_7_Dwn_Un

LDN   I_Support_1_Up
ST   I_I_Support_1_Up

LDN   I_Support_2_Up
ST   I_I_Support_2_Up

LDN   I_Support_3_Up
ST   I_I_Support_3_Up

LDN   I_Support_4_Up
ST   I_I_Support_4_Up

LDN   I_Support_5_Up
ST   I_I_Support_5_Up

LDN   I_Support_6_Up
ST   I_I_Support_6_Up

LDN   I_Support_7_Up
ST   I_I_Support_7_Up

LD   I_Support_1_Up_Un
AND  I_Support_1_Up_Un_aux    *AT %IW4.7;
ST   I_I_Support_1_Up_Un

LD   I_Support_2_Up_Un
ST   I_I_Support_2_Up_Un

LD   I_Support_3_Up_Un
ST   I_I_Support_3_Up_Un

LD   I_Support_4_Up_Un
ST   I_I_Support_4_Up_Un

LD   I_Support_5_Up_Un
ST   I_I_Support_5_Up_Un

LD   I_Support_6_Up_Un
ST   I_I_Support_6_Up_Un

LD   I_Support_7_Up_Un
ST   I_I_Support_7_Up_Un

*LD   I_MobileSpind_An
*ST   I_I_MobileSpind_An

*LD   I_FixedSpind_An
*ST   I_I_FixedSpind_An

LD   I_DistSens_Y
ST   I_I_DistSens_Y

LD   I_DistSens_Z
ST   I_I_DistSens_Z

LD   I_MobSpind_Y                              * Mobile spindle potentiometer sensor Y
ST   I_I_MobSpind_Y                            * Mobile spindle potentiometer sensor Y

LD   I_MobSpind_Z                              * Mobile spindle potentiometer sensor Z
ST   I_I_MobSpind_Z                            * Mobile spindle potentiometer sensor Z

LD   I_FixSpind_Y                              * Fixed spindle potentiometer sensor Y
ST   I_I_FixSpind_Y                            * Fixed spindle potentiometer sensor Y

LD   I_FixSpind_Z                              * Fixed spindle potentiometer sensor Z
ST   I_I_FixSpind_Z                            * Fixed spindle potentiometer sensor Z

LD   I_Pressure_Mobile
ST   I_I_Pressure_Mobile

LD   I_Pressure_Fix
ST   I_I_Pressure_Fix

LD   I_Loader_Reach_Pos
ST   I_I_Loader_Reach_Pos

LD   I_Loader_Back_Pos
ST   I_I_Loader_Back_Pos

LD   I_Loader_Alarm
ST   I_I_Loader_Alarm

LD   I_Mobile_Spindle_Slave_Open2
ST   I_I_Mobile_Spindle_Slave_Open2

LD   I_Flap_Home
ST   I_I_Flap_Home

*LD   I_Flap_Inclined
LD   O_O_Flap_Incline
ST   I_I_Flap_Inclined

LD   I_FlapL2_Home
ST   I_I_FlapL2_Home

*LD   I_FlapL2_Inclined
LD   O_O_FlapL2_Incline
ST   I_I_FlapL2_Inclined

LD   I_FlapL3_Home
ST   I_I_FlapL3_Home

*LD   I_FlapL3_Inclined
LD   O_O_FlapL3_Incline
ST   I_I_FlapL3_Inclined

*LD   I_FlapL4_Home
LD   O_O_FlapL4_Home
ST   I_I_FlapL4_Home

*LD   I_FlapL4_Inclined
LD   O_O_FlapL4_Incline
ST   I_I_FlapL4_Inclined

*LD   I_FlapL5_Home
LD   O_O_FlapL5_Home
ST   I_I_FlapL5_Home

*LD   I_FlapL5_Inclined
LD   O_O_FlapL5_Incline
ST   I_I_FlapL5_Inclined

LDN  I_M1_M2_M3_CLOSE
ST   I_I_M1_M2_M3_CLOSE

LDN  I_M1_M2_M3_OPEN
ST   I_I_M1_M2_M3_OPEN

LD   I_M1_M2_M3_ALARM
ST   I_I_M1_M2_M3_ALARM

LD   I_B1_B2_OPEN
ST   I_I_B1_B2_OPEN

LD   I_B1_B2_CLOSE
ST   I_I_B1_B2_CLOSE

LD   I_B1_B2_ALARM
ST   I_I_B1_B2_ALARM

LD   I_L1_Down
ST   I_I_L1_Down

*LD   I_Centering_Open
*LD   I_CenterZ1_Open
*AND  I_CenterZ2_Open
*AND  I_CenterZ3_Open
*AND  I_CenterZ4_Open
*ST   I_I_Centering_Open

* LD   I_Centering_Close
* ST   I_I_Centering_Close

LD   I_CenterZ1_Open
ST   I_I_Centering_Open_1

LD   I_CenterZ2_Open
ST   I_I_Centering_Open_2

LD   I_CenterZ3_Open
ST   I_I_Centering_Open_3

LD   I_CenterZ4_Open
ST   I_I_Centering_Open_4

LD   I_Detec_Weld
ST   I_I_Detec_Weld

LD   I_Pic_Weld
ST   I_I_Pic_Weld

LD   I_HomeChain_E
ST   I_I_HomeChain_E

LD   I_TubeOnChain_D_1
OR   I_TubeOnChain_D_2
OR   I_TubeOnChain_D_3
ST   I_I_TubeOnChain_D

LD   I_CylinderForw_F_1
AND  I_CylinderForw_F_2
AND  I_CylinderForw_F_3
ST   I_I_CylinderForw_F

LD   I_CylinderBack_F_1
AND  I_CylinderBack_F_2
AND  I_CylinderBack_F_3
ST   I_I_CylinderBack_F

LD   I_CylinderUp_G_1
AND  I_CylinderUp_G_2
AND  I_CylinderUp_G_3
ST   I_I_CylinderUp_G

LD   I_CylinderDwn_G_1
AND  I_CylinderDwn_G_2
AND  I_CylinderDwn_G_3
ST   I_I_CylinderDwn_G

LD   I_TubeOnSup_C_1
OR   I_TubeOnSup_C_2
ST   I_I_TubeOnSup_C

LDN  I_Loader_Slow
ST   I_I_Loader_Slow

LD   I_Bin_DoorUp
ST   I_I_Bin_DoorUp

*LD   I_Bin_DoorDwn
LD   O_O_Bin_Door
ST   I_I_Bin_DoorDwn

LDN  I_Photocell_Unload
AND  %cn0.rc8.0
S    %PLCmsg6.0

LDN  I_Photocell_Load
AND  %cn0.rc8.0
S    %PLCmsg6.1

*LD   I_Photocell_Reset
LD   Pul_Reset
OR   RESET_ALLARMI
R    %PLCmsg6.0
R    %PLCmsg6.1

LD   %PLCmsg6.0
OR   %PLCmsg6.1
ST   I_I_PHOTO_CELL
ST   PhotocellsOn

* LD   I_I_PHOTO_CELL
* AND  %PLCFLAGS.10
* ST   O_Luci_Photocell

LD   %LSRPlcOp1.28
JMPCN BYPASSPHCELL
      LD   0
      ST   PhotocellsOn
BYPASSPHCELL:

LD  I_SUPPORT_71_Dwn
ST  I_I_SUPPORT_71_Dwn

LD  I_SUPPORT_71_Up
ST  I_I_SUPPORT_71_Up

LD  I_SUPPORT_72_Dwn
ST  I_I_SUPPORT_72_Dwn

LD  I_SUPPORT_72_Up
ST  I_I_SUPPORT_72_Up

LD  I_SUPPORT_73_Dwn
ST  I_I_SUPPORT_73_Dwn

LD  I_SUPPORT_73_Up
ST  I_I_SUPPORT_73_Up

LD  I_SUPPORT_74_Dwn
ST  I_I_SUPPORT_74_Dwn

LD  I_SUPPORT_74_Up
ST  I_I_SUPPORT_74_Up

LD  I_SUPPORT_75_Dwn
ST  I_I_SUPPORT_75_Dwn

LD  I_SUPPORT_75_Up
ST  I_I_SUPPORT_75_Up

END_FUNCTION

FUNCTION  SHARED_MEMORY

LD   Pul_Reset                     ** (gPlc0.3)Reset pushbutton
ST   Reset                         ** Reset Command

LD   Pul_Start                     ** (gPlc0.1)Start pushbutton
ST   Start_Ch0                     ** Start Request to Ch0

LD   Pul_Stop
ST   Pul_Stop_Req

LD   PRGRUN_CN0
ST   ProgRunCh0                     * program in run ch0

*LD   ch7_in_jog
*ST   Ch7_Load_Jog

LD   I_I_EMERGENZA
ST   EmergButton

LD   EMER_GEN
ST   PlcEmerGen

LD   ch0_in_aut
ST   Ch0_Auto

LD   ch0_in_jog
ST   Ch0_Jog

LD   ch0_in_inc
ST   Ch0_Inc

LD   ch0_in_ref
ST   Ch0_Ref_Gen

LD   I_I_SEL_SINGLEREF
ST   Ch0_Ref_Sin

LD   Res_Ch0
ST   ResetChannels

LD   ChannelFeedrate
ST   MainChFeedrate

LD   Ch0InAlarm
ST   Ch0Alarm

LD   AxStopSincGRP
ST   AxStopSincGRPMacc

LD   Pon
ST   MainAxesPower

LD   GeneralCloseLoop
ST   MainAxesPowerAllowed

LD   Sel_Z_Ch8
ST   GstMaccSelZCh8

LD   Sel_Y_Ch8
ST   GstMaccSelYCh8

LD   Sel_U_Ch8
ST   GstMaccSelUCh8

LD   Sel_V_Ch8
ST   GstMaccSelVCh8

LD   Sel_W_Ch8
ST   GstMaccSelWCh8

LD   GrantPlcMoveX
ST   UsrGrantPlcMoveX

LD   GrantPlcMoveX1
ST   UsrGrantPlcMoveX1

END_FUNCTION

*******************************************************
* USER OUTPUT CONFIGURATION
*******************************************************

FUNCTION USR_OUT_CONFIG

* In case of emergency will cut off output of CNC by safety PLC
CAL  FTRIG_EMER(CLK=EMER_GEN)

LD   O_O_Mobile_Spindle_Slave_Open
ANDN FTRIG_EMER.Q
ST   Appoggio
CAL  TON_Spindle_Slave_Open_C2(IN=Appoggio,PT=4000)
LDN  TON_Spindle_Slave_Open_C2.Q
AND  O_O_Mobile_Spindle_Slave_Open
ST   SlaveSpdOpening
ST   O_Mobile_Spindle_Slave_Open

LD   O_O_Mobile_Spindle_Slave_Close
ANDN FTRIG_EMER.Q
ST   Appoggio
CAL  TON_Spindle_Slave_Close_C2(IN=Appoggio,PT=4000)
LDN  TON_Spindle_Slave_Close_C2.Q
AND  O_O_Mobile_Spindle_Slave_Close
ST   SlaveSpdClosing
ST   O_Mobile_Spindle_Slave_Close

LD   O_O_Mobile_Spindle_Open
ST   O_Mobile_Spindle_Open

LD   Invert_Mob_Spin_Open
ST   %PLCmsg8.8
JMPC Invert_Open
     LD   O_O_Mobile_Spindle_Close
     ST   O_Mobile_Spindle_Close

     LD   O_O_Mobile_Spindle_Open
     ST   O_Mobile_Spindle_Open
JMP  NO_Invert
Invert_Open:
     LD   O_O_Mobile_Spindle_Open
     ST   O_Mobile_Spindle_Close

     LD   O_O_Mobile_Spindle_Close
     ST   O_Mobile_Spindle_Open
NO_Invert:

LD   O_O_Mobile_Spindle_Slave_Brake
ST   O_Mobile_Spindle_Slave_Brake

LD   O_O_Ev_Support1_Up
ST   O_Ev_Support1_Up

LD   O_O_Ev_Support1_Dwn
ST   O_Ev_Support1_Dwn

LD   O_O_Ev_Support2_Up
ST   O_Ev_Support2_Up

LD   O_O_Ev_Support2_Dwn
ST   O_Ev_Support2_Dwn

LD   O_O_Ev_Support3_Up
ST   O_Ev_Support3_Up

LD   O_O_Ev_Support3_Dwn
ST   O_Ev_Support3_Dwn

LD   O_O_Ev_Support4_Up
ST   O_Ev_Support4_Up

LD   O_O_Ev_Support4_Dwn
ST   O_Ev_Support4_Dwn

LD   O_O_Ev_Support5_Up
ST   O_Ev_Support5_Up

LD   O_O_Ev_Support5_Dwn
ST   O_Ev_Support5_Dwn

LD   O_O_Ev_Support6_Up
ST   O_Ev_Support6_Up

LD   O_O_Ev_Support6_Dwn
ST   O_Ev_Support6_Dwn

LD   O_O_Ev_Support7_Up
ST   O_Ev_Support7_Up

LD   O_O_Ev_Support7_Dwn
ST   O_Ev_Support7_Dwn

LD   O_O_Ev_Support1_Up_Un
ST   O_Ev_Support1_Up_Un

LD   O_O_Ev_Support1_Dwn_Un
ST   O_Ev_Support1_Dwn_Un

LD   O_O_Ev_Support2_Up_Un
ST   O_Ev_Support2_Up_Un

LD   O_O_Ev_Support2_Dwn_Un
ST   O_Ev_Support2_Dwn_Un

LD   O_O_Ev_Support3_Up_Un
ST   O_Ev_Support3_Up_Un

LD   O_O_Ev_Support3_Dwn_Un
ST   O_Ev_Support3_Dwn_Un

LD   O_O_Ev_Support4_Up_Un
ST   O_Ev_Support4_Up_Un

LD   O_O_Ev_Support4_Dwn_Un
ST   O_Ev_Support4_Dwn_Un

LD   O_O_Ev_Support5_Up_Un
ST   O_Ev_Support5_Up_Un

LD   O_O_Ev_Support5_Dwn_Un
ST   O_Ev_Support5_Dwn_Un

LD   O_O_Ev_Support6_Up_Un
ST   O_Ev_Support6_Up_Un

LD   O_O_Ev_Support6_Dwn_Un
ST   O_Ev_Support6_Dwn_Un

LD   O_O_Ev_Support7_Up_Un
ST   O_Ev_Support7_Up_Un

LD   O_O_Ev_Support7_Dwn_Un
ST   O_Ev_Support7_Dwn_Un

LD   O_O_Pressure_Mobile
ST   O_Pressure_Mobile

LD   O_O_Pressure_MobileS
ST   O_Pressure_MobileS

LD   O_O_Loader_Back
ST   O_Loader_Back

LD   O_O_Bin_Door
ST   O_Bin_Door
STN  O_Bin_Door_Dwn

LD   O_O_FlapL2_Incline
ST   O_FlapL2_Incline

LD   O_O_FlapL2_Home
ST   O_FlapL2_Home

LD   I_Loader_Alarm
ST   %PLCerr21.18            ** Loader System Alarm

LD   O_O_Flap_Home
ST   O_Flap_Home

LD   O_O_Flap_Incline
ST   O_Flap_Incline

LD   O_O_SpindleFix_Open
ANDN FTRIG_EMER.Q
ST   Appoggio
CAL  TON_SpindleFix_Open_C1(IN=Appoggio,PT=4000)
LDN  TON_SpindleFix_Open_C1.Q
AND  O_O_SpindleFix_Open
ST   MidSpdOpening
ST   O_SpindleFix_Open

LD   O_O_SpindleFix_Close
ANDN FTRIG_EMER.Q
ST   Appoggio
CAL  TON_SpindleFix_Close_C1(IN=Appoggio,PT=4000)
LDN  TON_SpindleFix_Close_C1.Q
AND  O_O_SpindleFix_Close
ST   MidSpdClosing
ST   O_SpindleFix_Close

LD   O_O_FlapL3_Home
ST   O_FlapL3_Home

LD   O_O_FlapL3_Incline
ST   O_FlapL3_Incline

LD   O_O_FlapL4_Home
ST   O_FlapL4_Home

LD   O_O_FlapL4_Incline
ST   O_FlapL4_Incline

LD   O_O_FlapL5_Home
ST   O_FlapL5_Home

LD   O_O_FlapL5_Incline
ST   O_FlapL5_Incline

LD   O_O_M1_M2_M3_Open
ST   O_M1_M2_M3_Open

LD   O_O_M1_M2_M3_Close
ST   O_M1_M2_M3_Close

LD   O_O_Chain_Forw_D
ST   O_Chain_Forw_D

LD   O_O_Chain_Back_D
ST   O_Chain_Back_D

LD   O_O_Centering_Open_1
ST   O_Centering_Open_1

LD   O_O_Centering_Close_1
ST   O_Centering_Close_1

LD   O_O_Centering_Open_2
ST   O_Centering_Open_2

LD   O_O_Centering_Close_2
ST   O_Centering_Close_2

LD   O_O_Centering_Open_3
ST   O_Centering_Open_3

LD   O_O_Centering_Close_3
ST   O_Centering_Close_3

LD   O_O_Centering_Open_4
ST   O_Centering_Open_4

LD   O_O_Centering_Close_4
ST   O_Centering_Close_4

LD   O_O_B1_B2_Open
ST   O_B1_B2_Open

LD   O_O_B1_B2_Close
ST   O_B1_B2_Close

*************************************************
*  LOADER SUPPORTs
*************************************************
LD   O_O_CylinderUp_G
ST   O_CylinderUp_G

LD   O_O_CylinderDwn_G
ST   O_CylinderDwn_G

LD   O_O_CylinderForw_F
ST   O_CylinderForw_F

LD   O_O_CylinderBack_F
ST   O_CylinderBack_F

LD   O_O_Arm_Slow
ST   O_Arm_Slow

LD   O_O_Arm_Fast
ST   O_Arm_Fast

LD   O_O_Rst_InverterAlm
ST   O_Rst_InverterAlm

*************************************************
*  Weldseam Detection
*************************************************
LD   O_O_Detec_Weld_Piston
ST   O_Detec_Weld_Piston

LD   O_O_Detec_Weld
ST   O_Detec_Weld

LD   O_O_WeldDetec_En
OR   Btn_Weld_En               * Pulses
ST   O_WeldDetec_En

*************************************************
*  UNLOADER CYLINDERs
*************************************************
LD   O_O_Ev_Support72_Up
ST   O_Ev_Support72_Up

LD   O_O_Ev_Support72_Dwn
ST   O_Ev_Support72_Dwn

LD   O_O_Ev_Support71_Up
ST   O_Ev_Support71_Up

LD   O_O_Ev_Support71_Dwn
ST   O_Ev_Support71_Dwn

LD   O_O_Ev_Support73_Up
ST   O_Ev_Support73_Up

LD   O_O_Ev_Support73_Dwn
ST   O_Ev_Support73_Dwn

LD   O_O_Ev_Support74_Up
ST   O_Ev_Support74_Up

LD   O_O_Ev_Support74_Dwn
ST   O_Ev_Support74_Dwn

LD   O_O_Ev_Support75_Up
ST   O_Ev_Support75_Up

LD   O_O_Ev_Support75_Dwn
ST   O_Ev_Support75_Dwn

END_FUNCTION

(* ---- usrLatSu.plc ---- *)
#funcdec "FBSuppor.plc"
#funcdec "assi.plc"
#funcdec "DynMng.plc"
#funcdec "FBAux.plc"
#funcdec "SupForce.plc"
#funcdec "suppFB.plc"

VAR

* Axis support management

SUP1:               SUPPORT;
SUP2:               SUPPORT;
SUP3:               SUPPORT;
SUP4:               SUPPORT;

appoggio:              BOOL;
AdvOpen:              DWORD;

F_TRIG_RES_FOLL:     F_TRIG;

#include "iof.inc"
#include "usrIof.inc"
#include "cnc.inc"
END_VAR

VAR_IN_OUT
#include "usrIol.inc"
#include "mem.inc"
END_VAR

#include "Iol.inc"
#include "usrMem.inc"

FUNCTION LATERAL_SUPP

PATH  %cn9

*******************************************************
* Staggered avoidance position
* NOTE: IF %cn9.cc1.0 NOT DEFINED,
* THOSE AXES WILL BE HORIZONTAL RATHER THEN LATERAL
*******************************************************
LD   30000
ST   AdvOpen

LD   %ax30.ra0.0
JMPCN _closeloop_active
     LD   %ax30.ra92
     SUB  AdvOpen
     ST   PosUMis
JMP _no_loop
_closeloop_active:
     LD   %ax30.ra4
     ST   PosUMis
_no_loop:

*******************************************************
*         FOLLOWIING SUPPORTS MANAGEMENT              *
*******************************************************
 *(gIso49.0) Enable blendSwitch PLC writes (Lunette da ISO)
CAL  F_TRIG_RES_FOLL (CLK:=PRGRUN_CN0)
LD   F_TRIG_RES_FOLL.Q
OR   Pul_Reset
R    EnWriteBlendSwitch2
R    ParkAllLoadSuppCmd_LAT

LDN  PRGRUN_CN0
JMPCN RSTBLEND
     LD   %PLCFLAGS.0
	 ST   EnWriteBlendSwitch2
RSTBLEND:

LD   ALWAYS_ONE
ST   SUP1.xUaxDir
ST   SUP2.xUaxDir
ST   SUP3.xUaxDir
ST   SUP4.xUaxDir

LD   Reset
OR   EMER_GEN
ST   SUP1.xReset
ST   SUP2.xReset
ST   SUP3.xReset
ST   SUP4.xReset

LD   EnWriteBlendSwitch2
ST   SUP1.xBlendSwitchEn
ST   SUP2.xBlendSwitchEn
ST   SUP3.xBlendSwitchEn
ST   SUP4.xBlendSwitchEn

LD   OptEnabAutoParkLoad
ST   SUP1.xEnabAutoDwn
ST   SUP2.xEnabAutoDwn
ST   SUP3.xEnabAutoDwn
ST   SUP4.xEnabAutoDwn

LD   IN_M700_M704
EQ   704
OR   M700_BLEND
AND  %cn0.rc8.0
AND  O_O_Mobile_Spindle_Close
ANDN IN_M4_MODE
ST   SUP1.xEnabAutoUp
ST   SUP2.xEnabAutoUp
ST   SUP3.xEnabAutoUp
ST   SUP4.xEnabAutoUp

LD   IN_M700_M704
ST   SUP1.xM700_M704
ST   SUP2.xM700_M704
ST   SUP3.xM700_M704
ST   SUP4.xM700_M704

LD   IN_M4_MODE
JMPCN NOG1000PRK
     LD   0
     ST   SUP1.xM700_M704
     ST   SUP2.xM700_M704
     ST   SUP3.xM700_M704
     ST   SUP4.xM700_M704
NOG1000PRK:

LD   PosUMis
ST   SUP1.xSupervisePos
ST   SUP2.xSupervisePos
ST   SUP3.xSupervisePos
ST   SUP4.xSupervisePos

LD   OptForceLatOpen
ANDN (
LD   %gIso26
EQ   1
AND  NoRoundLatOpen
)
JMPCN FORCEOPENLAT
LD   0
ST   SUP1.xSupervisePos
ST   SUP2.xSupervisePos
ST   SUP3.xSupervisePos
ST   SUP4.xSupervisePos
FORCEOPENLAT:

LD   ParkingPosLoad_lat
ST   SUP1.xParkingPos
ST   SUP2.xParkingPos
ST   SUP3.xParkingPos
ST   SUP4.xParkingPos

LD   ThreshLoadingSupDown
ST   SUP1.xSuperviseOft
ST   SUP2.xSuperviseOft
ST   SUP3.xSuperviseOft
ST   SUP4.xSuperviseOft

LD   %ax30.ra3.0
ST   SUP1.xUaxStill
ST   SUP2.xUaxStill
ST   SUP3.xUaxStill
ST   SUP4.xUaxStill

* [lv, lat, ulv, uhor]=[0,1,2,3]
LD   1
ST   SUP1.xBlendId
ST   SUP2.xBlendId
ST   SUP3.xBlendId
ST   SUP4.xBlendId

* Support 1
LD   %cn9.cc1.1
JMPCN no_support_1

PATH  %ax81

LD   SUPPORT_1_Quota
ST   SUP1.xLimitSuppDwn

LD   ParkAllLoadSuppCmd_LAT
OR   Fun_M725_Ch0
OR   ParkUn51Sup_ISO
OR(
LD   Force_Open_Center_1
ANDN %cn0.rc8.0
AND  OptEnabAutoParkLoad
)
ST   SUP1.xParkCmd

CAL  SUP1

LD   SUP1.yReqGrant
ANDN ch9_in_ref
ST   usrReqGrantSupLat1

LD   SUP1.yHoldMovSupp
ANDN ch9_in_ref
ST   HoldO1SuppLoad_LAT

LD   SUP1.yHoldMovSuperv
ANDN ch9_in_ref
ANDN %cn9.cc1.0
ST   HoldO1Ax30_HOR

no_support_1:

* Support 2
LD   %cn9.cc1.2
JMPCN no_support_2

PATH  %ax82

LD   SUPPORT_2_Quota
ST   SUP2.xLimitSuppDwn

LD   ParkAllLoadSuppCmd_LAT
OR   Fun_M725_Ch0
OR   ParkUn52Sup_ISO
OR(
LD   Force_Open_Center_2
ANDN %cn0.rc8.0
AND  OptEnabAutoParkLoad
)
ST   SUP2.xParkCmd

CAL  SUP2

LD   SUP2.yReqGrant
ANDN ch9_in_ref
ST   usrReqGrantSupLat2

LD   SUP2.yHoldMovSupp
ANDN ch9_in_ref
ST   HoldO2SuppLoad_LAT

LD   SUP2.yHoldMovSuperv
ANDN ch9_in_ref
ANDN %cn9.cc1.0
ST   HoldO2Ax30_HOR

no_support_2:

* Support 3
LD   %cn9.cc1.3
JMPCN no_support_3

PATH  %ax83

LD   SUPPORT_3_Quota
ST   SUP3.xLimitSuppDwn

LD   ParkAllLoadSuppCmd_LAT
OR   Fun_M725_Ch0
OR   ParkUn53Sup_ISO
OR(
LD   Force_Open_Center_3
ANDN %cn0.rc8.0
AND  OptEnabAutoParkLoad
)
ST   SUP3.xParkCmd

CAL  SUP3

LD   SUP3.yReqGrant
ANDN ch9_in_ref
ST   usrReqGrantSupLat3

LD   SUP3.yHoldMovSupp
ANDN ch9_in_ref
ST   HoldO3SuppLoad_LAT

LD   SUP3.yHoldMovSuperv
ANDN ch9_in_ref
ANDN %cn9.cc1.0
ST   HoldO3Ax30_HOR

no_support_3:

* Support 4
LD   %cn9.cc1.4
JMPCN no_support_4

PATH  %ax84

LD   SUPPORT_4_Quota
ST   SUP4.xLimitSuppDwn

LD   ParkAllLoadSuppCmd_LAT
OR   Fun_M725_Ch0
OR   ParkUn54Sup_ISO
OR(
LD   Force_Open_Center_4
ANDN %cn0.rc8.0
AND  OptEnabAutoParkLoad
)
ST   SUP4.xParkCmd

CAL  SUP4

LD   SUP4.yReqGrant
ANDN ch9_in_ref
ST   usrReqGrantSupLat4

LD   SUP4.yHoldMovSupp
ANDN ch9_in_ref
ST   HoldO4SuppLoad_LAT

LD   SUP4.yHoldMovSuperv
ANDN ch9_in_ref
ANDN %cn9.cc1.0
ST   HoldO4Ax30_HOR

no_support_4:

END_FUNCTION
